LIN {X 0,Y 229.576,Z 730.403,A -85,B 0,C 180,E1 10386.317,E2 10386.317} C_VEL
LIN {X 0,Y 222.529,Z 739.722,A -85,B 0,C 180,E1 10381.712,E2 10381.712} C_VEL
LIN {X 0,Y 216.125,Z 748.376,A -85,B 0,C 180,E1 10376.069,E2 10376.069} C_VEL
LIN {X 0,Y 212.232,Z 754.139,A -85,B 0,C 180,E1 10371.117,E2 10371.117} C_VEL
LIN {X 0,Y 209.901,Z 758.178,A -85,B 0,C 180,E1 10366.605,E2 10366.605} C_VEL
LIN {X 0,Y 208.521,Z 761.292,A -85,B 0,C 180,E1 10361.898,E2 10361.898} C_VEL
LIN {X 0,Y 208.011,Z 763.279,A -85,B 0,C 180,E1 10357.456,E2 10357.456} C_VEL
LIN {X 0,Y 207.965,Z 764.362,A -85,B 0,C 180,E1 10353.031,E2 10353.031} C_VEL
LIN {X 0,Y 207.992,Z 764.571,A -85,B 0,C 180,E1 10348.898,E2 10348.898} C_VEL
LIN {X 0,Y 207.969,Z 763.727,A -85,B 0,C 180,E1 10343.929,E2 10343.929} C_VEL
LIN {X 0,Y 208.374,Z 761.739,A -85,B 0,C 180,E1 10338.935,E2 10338.935} C_VEL
LIN {X 0,Y 209.583,Z 758.806,A -85,B 0,C 180,E1 10334.223,E2 10334.223} C_VEL
LIN {X 0,Y 211.814,Z 754.811,A -85,B 0,C 180,E1 10329.557,E2 10329.557} C_VEL
LIN {X 0,Y 215.171,Z 749.706,A -85,B 0,C 180,E1 10324.98,E2 10324.98} C_VEL
LIN {X 0,Y 219.672,Z 743.459,A -85,B 0,C 180,E1 10320.559,E2 10320.559} C_VEL
LIN {X 0,Y 225.328,Z 735.97,A -85,B 0,C 180,E1 10316.316,E2 10316.316} C_VEL
LIN {X 0,Y 233.394,Z 725.524,A -85,B 0,C 180,E1 10311.603,E2 10311.603} C_VEL
LIN {X 0,Y 242.359,Z 713.434,A -85,B 0,C 180,E1 10307.428,E2 10307.428} C_VEL
LIN {X 0,Y 250.273,Z 702.419,A -85,B 0,C 180,E1 10304.353,E2 10304.353} C_VEL
LIN {X 0,Y 258.267,Z 690.731,A -85,B 0,C 180,E1 10301.66,E2 10301.66} C_VEL
LIN {X 0,Y 266.491,Z 677.953,A -85,B 0,C 180,E1 10299.223,E2 10299.223} C_VEL
LIN {X 0,Y 274.84,Z 663.987,A -85,B 0,C 180,E1 10297.018,E2 10297.018} C_VEL
LIN {X 0,Y 285.068,Z 645.138,A -85,B 0,C 180,E1 10294.627,E2 10294.627} C_VEL
LIN {X 0,Y 293.059,Z 628.408,A -85,B 0,C 180,E1 10292.943,E2 10292.943} C_VEL
LIN {X 0,Y 299.949,Z 612.279,A -85,B 0,C 180,E1 10291.614,E2 10291.614} C_VEL
LIN {X 0,Y 305.879,Z 596.561,A -85,B 0,C 180,E1 10290.544,E2 10290.544} C_VEL
LIN {X 0,Y 311.16,Z 580.497,A -85,B 0,C 180,E1 10289.644,E2 10289.644} C_VEL
LIN {X 0,Y 315.755,Z 564.123,A -85,B 0,C 180,E1 10288.9,E2 10288.9} C_VEL
LIN {X 0,Y 319.912,Z 546.219,A -85,B 0,C 180,E1 10288.263,E2 10288.263} C_VEL
LIN {X 0,Y 323.86,Z 523.655,A -85,B 0,C 180,E1 10287.653,E2 10287.653} C_VEL
LIN {X 0,Y 327.226,Z 489.016,A -85,B 0,C 180,E1 10286.991,E2 10286.991} C_VEL
LIN {X 0,Y 336.453,Z 381.786,A -85,B 0,C 180,E1 10285.079,E2 10285.079} C_VEL
LIN {X 0,Y 331.591,Z 370.301,A -85,B 0,C 180,E1 10282.611,E2 10282.611} C_VEL
LIN {X 0,Y 328.158,Z 363.719,A -85,B 0,C 180,E1 10280.745,E2 10280.745} C_VEL
LIN {X 0,Y 323.384,Z 355.371,A -85,B 0,C 180,E1 10277.825,E2 10277.825} C_VEL
LIN {X 0,Y 319.206,Z 348.74,A -85,B 0,C 180,E1 10274.791,E2 10274.791} C_VEL
LIN {X 0,Y 317.453,Z 345.951,A -85,B 0,C 180,E1 10273.293,E2 10273.293} C_VEL
LIN {X 0,Y 315.139,Z 342.181,A -85,B 0,C 180,E1 10270.975,E2 10270.975} C_VEL
LIN {X 0,Y 312.623,Z 337.855,A -85,B 0,C 180,E1 10267.628,E2 10267.628} C_VEL
LIN {X 0,Y 310.185,Z 334.373,A -85,B 0,C 180,E1 10260.369,E2 10260.369} C_VEL
LIN {X 0,Y 310.304,Z 334.935,A -85,B 0,C 180,E1 10257.784,E2 10257.784} C_VEL
LIN {X 0,Y 312.654,Z 337.983,A -85,B 0,C 180,E1 10252.003,E2 10252.003} C_VEL
LIN {X 0,Y 315.196,Z 342.253,A -85,B 0,C 180,E1 10248.657,E2 10248.657} C_VEL
LIN {X 0,Y 318.856,Z 348.121,A -85,B 0,C 180,E1 10245.192,E2 10245.192} C_VEL
LIN {X 0,Y 322.317,Z 353.748,A -85,B 0,C 180,E1 10242.581,E2 10242.581} C_VEL
LIN {X 0,Y 326.66,Z 361.098,A -85,B 0,C 180,E1 10239.811,E2 10239.811} C_VEL
LIN {X 0,Y 332.388,Z 371.39,A -85,B 0,C 180,E1 10236.698,E2 10236.698} C_VEL
LIN {X 0,Y 346.546,Z 396.133,A -85,B 0,C 180,E1 10230.674,E2 10230.674} C_VEL
LIN {X 0,Y 360.991,Z 413.89,A -85,B 0,C 180,E1 10226.169,E2 10226.169} C_VEL
LIN {X 0,Y 383.3,Z 434.199,A -85,B 0,C 180,E1 10220.855,E2 10220.855} C_VEL
LIN {X 0,Y 397.073,Z 444.864,A -85,B 0,C 180,E1 10218.092,E2 10218.092} C_VEL
LIN {X 0,Y 406.656,Z 452.456,A -85,B 0,C 180,E1 10216.052,E2 10216.052} C_VEL
LIN {X 0,Y 416.596,Z 460.43,A -85,B 0,C 180,E1 10213.743,E2 10213.743} C_VEL
LIN {X 0,Y 425.756,Z 468.037,A -85,B 0,C 180,E1 10211.379,E2 10211.379} C_VEL
LIN {X 0,Y 433.593,Z 474.542,A -85,B 0,C 180,E1 10209.181,E2 10209.181} C_VEL
LIN {X 0,Y 443.165,Z 482.341,A -85,B 0,C 180,E1 10206.343,E2 10206.343} C_VEL
LIN {X 0,Y 451.87,Z 489.268,A -85,B 0,C 180,E1 10203.637,E2 10203.637} C_VEL
LIN {X 0,Y 459.287,Z 495.387,A -85,B 0,C 180,E1 10201.176,E2 10201.176} C_VEL
LIN {X 0,Y 464.734,Z 499.578,A -85,B 0,C 180,E1 10199.269,E2 10199.269} C_VEL
LIN {X 0,Y 471.201,Z 504.679,A -85,B 0,C 180,E1 10196.867,E2 10196.867} C_VEL
LIN {X 0,Y 476.22,Z 508.342,A -85,B 0,C 180,E1 10194.9,E2 10194.9} C_VEL
LIN {X 0,Y 481.698,Z 512.833,A -85,B 0,C 180,E1 10192.524,E2 10192.524} C_VEL
LIN {X 0,Y 487.412,Z 516.593,A -85,B 0,C 180,E1 10189.844,E2 10189.844} C_VEL
LIN {X 0,Y 491.994,Z 520.595,A -85,B 0,C 180,E1 10187.38,E2 10187.38} C_VEL
LIN {X 0,Y 496.009,Z 523.409,A -85,B 0,C 180,E1 10184.951,E2 10184.951} C_VEL
LIN {X 0,Y 499.622,Z 525.352,A -85,B 0,C 180,E1 10182.41,E2 10182.41} C_VEL
LIN {X 0,Y 501.043,Z 526.363,A -85,B 0,C 180,E1 10181.276,E2 10181.276} C_VEL
LIN {X 0,Y 503.296,Z 528.639,A -85,B 0,C 180,E1 10179.029,E2 10179.029} C_VEL
LIN {X 0,Y 505.299,Z 530.408,A -85,B 0,C 180,E1 10176.59,E2 10176.59} C_VEL
LIN {X 0,Y 506.622,Z 531.453,A -85,B 0,C 180,E1 10174.074,E2 10174.074} C_VEL
LIN {X 0,Y 507.429,Z 531.971,A -85,B 0,C 180,E1 10171.468,E2 10171.468} C_VEL
LIN {X 0,Y 507.45,Z 531.985,A -85,B 0,C 180,E1 10169.097,E2 10169.097} C_VEL
LIN {X 0,Y 506.956,Z 531.659,A -85,B 0,C 180,E1 10166.608,E2 10166.608} C_VEL
LIN {X 0,Y 505.654,Z 530.72,A -85,B 0,C 180,E1 10164.068,E2 10164.068} C_VEL
LIN {X 0,Y 503.867,Z 529.16,A -85,B 0,C 180,E1 10161.557,E2 10161.557} C_VEL
LIN {X 0,Y 501.524,Z 526.933,A -85,B 0,C 180,E1 10159.2,E2 10159.2} C_VEL
LIN {X 0,Y 500.006,Z 525.51,A -85,B 0,C 180,E1 10157.881,E2 10157.881} C_VEL
LIN {X 0,Y 496.616,Z 523.748,A -85,B 0,C 180,E1 10155.425,E2 10155.425} C_VEL
LIN {X 0,Y 492.566,Z 521.055,A -85,B 0,C 180,E1 10152.963,E2 10152.963} C_VEL
LIN {X 0,Y 488.034,Z 517.174,A -85,B 0,C 180,E1 10150.469,E2 10150.469} C_VEL
LIN {X 0,Y 484.075,Z 514.456,A -85,B 0,C 180,E1 10148.558,E2 10148.558} C_VEL
LIN {X 0,Y 478.527,Z 510.37,A -85,B 0,C 180,E1 10146.089,E2 10146.089} C_VEL
LIN {X 0,Y 473.228,Z 506.031,A -85,B 0,C 180,E1 10143.895,E2 10143.895} C_VEL
LIN {X 0,Y 466.718,Z 501.246,A -85,B 0,C 180,E1 10141.448,E2 10141.448} C_VEL
LIN {X 0,Y 461.036,Z 496.657,A -85,B 0,C 180,E1 10139.431,E2 10139.431} C_VEL
LIN {X 0,Y 453.633,Z 490.858,A -85,B 0,C 180,E1 10136.95,E2 10136.95} C_VEL
LIN {X 0,Y 446.485,Z 485.103,A -85,B 0,C 180,E1 10134.678,E2 10134.678} C_VEL
LIN {X 0,Y 437.683,Z 477.869,A -85,B 0,C 180,E1 10132.014,E2 10132.014} C_VEL
LIN {X 0,Y 428.629,Z 470.268,A -85,B 0,C 180,E1 10129.402,E2 10129.402} C_VEL
LIN {X 0,Y 420.998,Z 464.055,A -85,B 0,C 180,E1 10127.364,E2 10127.364} C_VEL
LIN {X 0,Y 411.623,Z 456.502,A -85,B 0,C 180,E1 10125.08,E2 10125.08} C_VEL
LIN {X 0,Y 401.509,Z 448.491,A -85,B 0,C 180,E1 10122.833,E2 10122.833} C_VEL
LIN {X 0,Y 390.28,Z 439.766,A -85,B 0,C 180,E1 10120.55,E2 10120.55} C_VEL
LIN {X 0,Y 363.524,Z 416.49,A -85,B 0,C 180,E1 10114.514,E2 10114.514} C_VEL
LIN {X 0,Y 349.69,Z 400.357,A -85,B 0,C 180,E1 10110.405,E2 10110.405} C_VEL
LIN {X 0,Y 339.201,Z 384.437,A -85,B 0,C 180,E1 10106.478,E2 10106.478} C_VEL
LIN {X 0,Y 331.747,Z 370.145,A -85,B 0,C 180,E1 10102.974,E2 10102.974} C_VEL
LIN {X 0,Y 325.408,Z 358.84,A -85,B 0,C 180,E1 10099.428,E2 10099.428} C_VEL
LIN {X 0,Y 320.76,Z 351.104,A -85,B 0,C 180,E1 10096.293,E2 10096.293} C_VEL
LIN {X 0,Y 317.522,Z 346.047,A -85,B 0,C 180,E1 10093.661,E2 10093.661} C_VEL
LIN {X 0,Y 315.196,Z 342.25,A -85,B 0,C 180,E1 10091.343,E2 10091.343} C_VEL
LIN {X 0,Y 312.654,Z 337.981,A -85,B 0,C 180,E1 10087.997,E2 10087.997} C_VEL
LIN {X 0,Y 310.184,Z 334.34,A -85,B 0,C 180,E1 10080.554,E2 10080.554} C_VEL
LIN {X 0,Y 310.42,Z 335.246,A -85,B 0,C 180,E1 10077.415,E2 10077.415} C_VEL
LIN {X 0,Y 312.674,Z 338,A -85,B 0,C 180,E1 10072.281,E2 10072.281} C_VEL
LIN {X 0,Y 315.139,Z 342.183,A -85,B 0,C 180,E1 10069.025,E2 10069.025} C_VEL
LIN {X 0,Y 318.785,Z 347.988,A -85,B 0,C 180,E1 10065.56,E2 10065.56} C_VEL
LIN {X 0,Y 322.733,Z 354.42,A -85,B 0,C 180,E1 10062.604,E2 10062.604} C_VEL
LIN {X 0,Y 327.577,Z 362.616,A -85,B 0,C 180,E1 10059.59,E2 10059.59} C_VEL
LIN {X 0,Y 331.359,Z 369.794,A -85,B 0,C 180,E1 10057.513,E2 10057.513} C_VEL
LIN {X 0,Y 335.907,Z 380.499,A -85,B 0,C 180,E1 10055.183,E2 10055.183} C_VEL
LIN {X 0,Y 336.48,Z 382.275,A -85,B 0,C 180,E1 10054.888,E2 10054.888} C_VEL
LIN {X 0,Y 324.566,Z 517.418,A -85,B 0,C 180,E1 10052.477,E2 10052.477} C_VEL
LIN {X 0,Y 321.459,Z 538.537,A -85,B 0,C 180,E1 10051.966,E2 10051.966} C_VEL
LIN {X 0,Y 316.405,Z 561.647,A -85,B 0,C 180,E1 10051.199,E2 10051.199} C_VEL
LIN {X 0,Y 311.542,Z 579.253,A -85,B 0,C 180,E1 10050.418,E2 10050.418} C_VEL
LIN {X 0,Y 306.252,Z 595.5,A -85,B 0,C 180,E1 10049.522,E2 10049.522} C_VEL
LIN {X 0,Y 300.315,Z 611.359,A -85,B 0,C 180,E1 10048.455,E2 10048.455} C_VEL
LIN {X 0,Y 300.203,Z 611.641,A -85,B 0,C 180,E1 10048.434,E2 10048.434} C_VEL
LIN {X 0,Y 296.909,Z 618.594,A -85,B 0,C 180,E1 10048.072,E2 10048.072} C_VEL
LIN {X 0,Y 285.993,Z 635.3,A -85,B 0,C 180,E1 10047.577,E2 10047.577} C_VEL
LIN {X 0,Y 282.279,Z 641.505,A -85,B 0,C 180,E1 10047.099,E2 10047.099} C_VEL
LIN {X 0,Y 273.798,Z 657.322,A -85,B 0,C 180,E1 10045.242,E2 10045.242} C_VEL
LIN {X 0,Y 263.053,Z 675.28,A -85,B 0,C 180,E1 10042.591,E2 10042.591} C_VEL
LIN {X 0,Y 254.155,Z 688.774,A -85,B 0,C 180,E1 10040.09,E2 10040.09} C_VEL
LIN {X 0,Y 245.788,Z 700.659,A -85,B 0,C 180,E1 10037.411,E2 10037.411} C_VEL
LIN {X 0,Y 237.997,Z 711.151,A -85,B 0,C 180,E1 10034.549,E2 10034.549} C_VEL
LIN {X 0,Y 230.344,Z 721.041,A -85,B 0,C 180,E1 10031.278,E2 10031.278} C_VEL
LIN {X 0,Y 223.04,Z 730.224,A -85,B 0,C 180,E1 10027.561,E2 10027.561} C_VEL
LIN {X 0,Y 215.613,Z 739.544,A -85,B 0,C 180,E1 10022.854,E2 10022.854} C_VEL
LIN {X 0,Y 208.793,Z 748.224,A -85,B 0,C 180,E1 10017.033,E2 10017.033} C_VEL
LIN {X 0,Y 204.742,Z 753.82,A -85,B 0,C 180,E1 10012.085,E2 10012.085} C_VEL
LIN {X 0,Y 202.12,Z 758,A -85,B 0,C 180,E1 10007.264,E2 10007.264} C_VEL
LIN {X 0,Y 200.59,Z 761.149,A -85,B 0,C 180,E1 10002.308,E2 10002.308} C_VEL
LIN {X 0,Y 200.012,Z 763.193,A -85,B 0,C 180,E1 9997.467,E2 9997.467} C_VEL
LIN {X 0,Y 199.965,Z 764.187,A -85,B 0,C 180,E1 9993.153,E2 9993.153} C_VEL
LIN {X 0,Y 199.993,Z 764.396,A -85,B 0,C 180,E1 9988.854,E2 9988.854} C_VEL
LIN {X 0,Y 199.969,Z 763.641,A -85,B 0,C 180,E1 9983.973,E2 9983.973} C_VEL
LIN {X 0,Y 200.391,Z 761.712,A -85,B 0,C 180,E1 9978.78,E2 9978.78} C_VEL
LIN {X 0,Y 201.775,Z 758.628,A -85,B 0,C 180,E1 9973.595,E2 9973.595} C_VEL
LIN {X 0,Y 204.194,Z 754.633,A -85,B 0,C 180,E1 9968.758,E2 9968.758} C_VEL
LIN {X 0,Y 207.791,Z 749.536,A -85,B 0,C 180,E1 9964.034,E2 9964.034} C_VEL
LIN {X 0,Y 212.273,Z 743.68,A -85,B 0,C 180,E1 9959.739,E2 9959.739} C_VEL
LIN {X 0,Y 217.804,Z 736.729,A -85,B 0,C 180,E1 9955.626,E2 9955.626} C_VEL
LIN {X 0,Y 224.59,Z 728.288,A -85,B 0,C 180,E1 9951.589,E2 9951.589} C_VEL
LIN {X 0,Y 233.32,Z 717.328,A -85,B 0,C 180,E1 9947.389,E2 9947.389} C_VEL
LIN {X 0,Y 243.507,Z 703.824,A -85,B 0,C 180,E1 9943.39,E2 9943.39} C_VEL
LIN {X 0,Y 252.319,Z 691.443,A -85,B 0,C 180,E1 9940.469,E2 9940.469} C_VEL
LIN {X 0,Y 260.46,Z 679.274,A -85,B 0,C 180,E1 9938.106,E2 9938.106} C_VEL
LIN {X 0,Y 268.349,Z 666.612,A -85,B 0,C 180,E1 9936.055,E2 9936.055} C_VEL
LIN {X 0,Y 276.069,Z 653.203,A -85,B 0,C 180,E1 9934.244,E2 9934.244} C_VEL
LIN {X 0,Y 283.669,Z 638.754,A -85,B 0,C 180,E1 9932.614,E2 9932.614} C_VEL
LIN {X 0,Y 291.329,Z 622.592,A -85,B 0,C 180,E1 9931.106,E2 9931.106} C_VEL
LIN {X 0,Y 299.967,Z 601.695,A -85,B 0,C 180,E1 9929.555,E2 9929.555} C_VEL
LIN {X 0,Y 306.486,Z 582.805,A -85,B 0,C 180,E1 9928.465,E2 9928.465} C_VEL
LIN {X 0,Y 311.362,Z 566.176,A -85,B 0,C 180,E1 9927.699,E2 9927.699} C_VEL
LIN {X 0,Y 315.623,Z 548.674,A -85,B 0,C 180,E1 9927.066,E2 9927.066} C_VEL
LIN {X 0,Y 318.97,Z 531.138,A -85,B 0,C 180,E1 9926.574,E2 9926.574} C_VEL
LIN {X 0,Y 321.456,Z 512.557,A -85,B 0,C 180,E1 9926.159,E2 9926.159} C_VEL
LIN {X 0,Y 332.773,Z 385.796,A -85,B 0,C 180,E1 9923.908,E2 9923.908} C_VEL
LIN {X 0,Y 328.392,Z 375.154,A -85,B 0,C 180,E1 9921.525,E2 9921.525} C_VEL
LIN {X 0,Y 323.343,Z 365.828,A -85,B 0,C 180,E1 9918.526,E2 9918.526} C_VEL
LIN {X 0,Y 318.985,Z 358.378,A -85,B 0,C 180,E1 9915.453,E2 9915.453} C_VEL
LIN {X 0,Y 316.074,Z 353.64,A -85,B 0,C 180,E1 9912.98,E2 9912.98} C_VEL
LIN {X 0,Y 313.829,Z 349.888,A -85,B 0,C 180,E1 9910.649,E2 9910.649} C_VEL
LIN {X 0,Y 311.244,Z 345.447,A -85,B 0,C 180,E1 9907.012,E2 9907.012} C_VEL
LIN {X 0,Y 309.204,Z 342.3,A -85,B 0,C 180,E1 9900.185,E2 9900.185} C_VEL
LIN {X 0,Y 309.417,Z 343.167,A -85,B 0,C 180,E1 9897.222,E2 9897.222} C_VEL
LIN {X 0,Y 311.549,Z 345.958,A -85,B 0,C 180,E1 9892.16,E2 9892.16} C_VEL
LIN {X 0,Y 314.625,Z 351.207,A -85,B 0,C 180,E1 9888.162,E2 9888.162} C_VEL
LIN {X 0,Y 317.538,Z 356.047,A -85,B 0,C 180,E1 9885.409,E2 9885.409} C_VEL
LIN {X 0,Y 320.818,Z 361.511,A -85,B 0,C 180,E1 9882.871,E2 9882.871} C_VEL
LIN {X 0,Y 325.497,Z 369.707,A -85,B 0,C 180,E1 9879.829,E2 9879.829} C_VEL
LIN {X 0,Y 331.416,Z 380.885,A -85,B 0,C 180,E1 9876.578,E2 9876.578} C_VEL
LIN {X 0,Y 342.541,Z 401.036,A -85,B 0,C 180,E1 9871.683,E2 9871.683} C_VEL
LIN {X 0,Y 356.013,Z 418.443,A -85,B 0,C 180,E1 9867.224,E2 9867.224} C_VEL
LIN {X 0,Y 373.061,Z 435.003,A -85,B 0,C 180,E1 9862.815,E2 9862.815} C_VEL
LIN {X 0,Y 393.784,Z 451.72,A -85,B 0,C 180,E1 9858.492,E2 9858.492} C_VEL
LIN {X 0,Y 404.068,Z 459.754,A -85,B 0,C 180,E1 9856.338,E2 9856.338} C_VEL
LIN {X 0,Y 413.478,Z 467.249,A -85,B 0,C 180,E1 9854.192,E2 9854.192} C_VEL
LIN {X 0,Y 422.851,Z 474.87,A -85,B 0,C 180,E1 9851.853,E2 9851.853} C_VEL
LIN {X 0,Y 431.409,Z 481.9,A -85,B 0,C 180,E1 9849.484,E2 9849.484} C_VEL
LIN {X 0,Y 441.106,Z 489.743,A -85,B 0,C 180,E1 9846.636,E2 9846.636} C_VEL
LIN {X 0,Y 449.6,Z 496.451,A -85,B 0,C 180,E1 9844.006,E2 9844.006} C_VEL
LIN {X 0,Y 457.074,Z 502.656,A -85,B 0,C 180,E1 9841.551,E2 9841.551} C_VEL
LIN {X 0,Y 463.048,Z 507.191,A -85,B 0,C 180,E1 9839.49,E2 9839.49} C_VEL
LIN {X 0,Y 469.743,Z 512.437,A -85,B 0,C 180,E1 9837.026,E2 9837.026} C_VEL
LIN {X 0,Y 474.826,Z 516.148,A -85,B 0,C 180,E1 9835.037,E2 9835.037} C_VEL
LIN {X 0,Y 480.395,Z 520.663,A -85,B 0,C 180,E1 9832.644,E2 9832.644} C_VEL
LIN {X 0,Y 486.164,Z 524.446,A -85,B 0,C 180,E1 9829.96,E2 9829.96} C_VEL
LIN {X 0,Y 490.743,Z 528.395,A -85,B 0,C 180,E1 9827.531,E2 9827.531} C_VEL
LIN {X 0,Y 494.745,Z 531.223,A -85,B 0,C 180,E1 9825.11,E2 9825.11} C_VEL
LIN {X 0,Y 498.505,Z 533.242,A -85,B 0,C 180,E1 9822.509,E2 9822.509} C_VEL
LIN {X 0,Y 500.029,Z 534.336,A -85,B 0,C 180,E1 9821.3,E2 9821.3} C_VEL
LIN {X 0,Y 502.292,Z 536.591,A -85,B 0,C 180,E1 9819.047,E2 9819.047} C_VEL
LIN {X 0,Y 504.312,Z 538.351,A -85,B 0,C 180,E1 9816.602,E2 9816.602} C_VEL
LIN {X 0,Y 505.641,Z 539.394,A -85,B 0,C 180,E1 9814.082,E2 9814.082} C_VEL
LIN {X 0,Y 506.453,Z 539.911,A -85,B 0,C 180,E1 9811.471,E2 9811.471} C_VEL
LIN {X 0,Y 506.474,Z 539.925,A -85,B 0,C 180,E1 9809.095,E2 9809.095} C_VEL
LIN {X 0,Y 505.979,Z 539.6,A -85,B 0,C 180,E1 9806.602,E2 9806.602} C_VEL
LIN {X 0,Y 504.686,Z 538.676,A -85,B 0,C 180,E1 9804.088,E2 9804.088} C_VEL
LIN {X 0,Y 502.973,Z 537.211,A -85,B 0,C 180,E1 9801.657,E2 9801.657} C_VEL
LIN {X 0,Y 500.51,Z 534.898,A -85,B 0,C 180,E1 9799.178,E2 9799.178} C_VEL
LIN {X 0,Y 498.821,Z 533.377,A -85,B 0,C 180,E1 9797.734,E2 9797.734} C_VEL
LIN {X 0,Y 495.316,Z 531.539,A -85,B 0,C 180,E1 9795.23,E2 9795.23} C_VEL
LIN {X 0,Y 491.354,Z 528.893,A -85,B 0,C 180,E1 9792.841,E2 9792.841} C_VEL
LIN {X 0,Y 486.699,Z 524.95,A -85,B 0,C 180,E1 9790.313,E2 9790.313} C_VEL
LIN {X 0,Y 481.953,Z 521.71,A -85,B 0,C 180,E1 9788.03,E2 9788.03} C_VEL
LIN {X 0,Y 476.405,Z 517.535,A -85,B 0,C 180,E1 9785.629,E2 9785.629} C_VEL
LIN {X 0,Y 471.685,Z 513.736,A -85,B 0,C 180,E1 9783.706,E2 9783.706} C_VEL
LIN {X 0,Y 465.205,Z 508.978,A -85,B 0,C 180,E1 9781.275,E2 9781.275} C_VEL
LIN {X 0,Y 459.27,Z 504.242,A -85,B 0,C 180,E1 9779.191,E2 9779.191} C_VEL
LIN {X 0,Y 451.846,Z 498.442,A -85,B 0,C 180,E1 9776.721,E2 9776.721} C_VEL
LIN {X 0,Y 443.612,Z 491.846,A -85,B 0,C 180,E1 9774.13,E2 9774.13} C_VEL
LIN {X 0,Y 435.125,Z 484.929,A -85,B 0,C 180,E1 9771.591,E2 9771.591} C_VEL
LIN {X 0,Y 426.196,Z 477.515,A -85,B 0,C 180,E1 9769.064,E2 9769.064} C_VEL
LIN {X 0,Y 418.744,Z 471.473,A -85,B 0,C 180,E1 9767.094,E2 9767.094} C_VEL
LIN {X 0,Y 408.582,Z 463.367,A -85,B 0,C 180,E1 9764.666,E2 9764.666} C_VEL
LIN {X 0,Y 398.159,Z 455.228,A -85,B 0,C 180,E1 9762.408,E2 9762.408} C_VEL
LIN {X 0,Y 385.414,Z 445.344,A -85,B 0,C 180,E1 9759.852,E2 9759.852} C_VEL
LIN {X 0,Y 360.455,Z 423.252,A -85,B 0,C 180,E1 9754.032,E2 9754.032} C_VEL
LIN {X 0,Y 346.851,Z 407.086,A -85,B 0,C 180,E1 9749.868,E2 9749.868} C_VEL
LIN {X 0,Y 336.504,Z 391.004,A -85,B 0,C 180,E1 9745.852,E2 9745.852} C_VEL
LIN {X 0,Y 329.357,Z 376.881,A -85,B 0,C 180,E1 9742.349,E2 9742.349} C_VEL
LIN {X 0,Y 323.439,Z 365.989,A -85,B 0,C 180,E1 9738.895,E2 9738.895} C_VEL
LIN {X 0,Y 319.067,Z 358.487,A -85,B 0,C 180,E1 9735.821,E2 9735.821} C_VEL
LIN {X 0,Y 315.948,Z 353.458,A -85,B 0,C 180,E1 9733.171,E2 9733.171} C_VEL
LIN {X 0,Y 313.885,Z 349.959,A -85,B 0,C 180,E1 9731.019,E2 9731.019} C_VEL
LIN {X 0,Y 311.282,Z 345.481,A -85,B 0,C 180,E1 9727.382,E2 9727.382} C_VEL
LIN {X 0,Y 309.204,Z 342.276,A -85,B 0,C 180,E1 9720.37,E2 9720.37} C_VEL
LIN {X 0,Y 309.521,Z 343.402,A -85,B 0,C 180,E1 9717.037,E2 9717.037} C_VEL
LIN {X 0,Y 311.518,Z 345.832,A -85,B 0,C 180,E1 9712.531,E2 9712.531} C_VEL
LIN {X 0,Y 313.996,Z 350.073,A -85,B 0,C 180,E1 9709.171,E2 9709.171} C_VEL
LIN {X 0,Y 317.365,Z 355.729,A -85,B 0,C 180,E1 9705.867,E2 9705.867} C_VEL
LIN {X 0,Y 321.608,Z 362.734,A -85,B 0,C 180,E1 9702.634,E2 9702.634} C_VEL
LIN {X 0,Y 326.414,Z 371.468,A -85,B 0,C 180,E1 9699.591,E2 9699.591} C_VEL
LIN {X 0,Y 329.354,Z 377.369,A -85,B 0,C 180,E1 9697.933,E2 9697.933} C_VEL
LIN {X 0,Y 332.795,Z 386.105,A -85,B 0,C 180,E1 9696.068,E2 9696.068} C_VEL
LIN {X 0,Y 320.935,Z 517.284,A -85,B 0,C 180,E1 9693.746,E2 9693.746} C_VEL
LIN {X 0,Y 317.72,Z 538.657,A -85,B 0,C 180,E1 9693.235,E2 9693.235} C_VEL
LIN {X 0,Y 312.796,Z 560.808,A -85,B 0,C 180,E1 9692.513,E2 9692.513} C_VEL
LIN {X 0,Y 307.654,Z 579.077,A -85,B 0,C 180,E1 9691.72,E2 9691.72} C_VEL
LIN {X 0,Y 302.248,Z 595.324,A -85,B 0,C 180,E1 9690.837,E2 9690.837} C_VEL
LIN {X 0,Y 296.176,Z 611.183,A -85,B 0,C 180,E1 9689.784,E2 9689.784} C_VEL
LIN {X 0,Y 289.48,Z 626.62,A -85,B 0,C 180,E1 9688.544,E2 9688.544} C_VEL
LIN {X 0,Y 282.279,Z 641.505,A -85,B 0,C 180,E1 9687.099,E2 9687.099} C_VEL
LIN {X 0,Y 278.481,Z 647.851,A -85,B 0,C 180,E1 9686.583,E2 9686.583} C_VEL
LIN {X 0,Y 266.227,Z 663.246,A -85,B 0,C 180,E1 9685.662,E2 9685.662} C_VEL
LIN {X 0,Y 262.112,Z 668.947,A -85,B 0,C 180,E1 9684.998,E2 9684.998} C_VEL
LIN {X 0,Y 250.948,Z 685.928,A -85,B 0,C 180,E1 9682.075,E2 9682.075} C_VEL
LIN {X 0,Y 240.863,Z 699.801,A -85,B 0,C 180,E1 9679.012,E2 9679.012} C_VEL
LIN {X 0,Y 232.81,Z 710.272,A -85,B 0,C 180,E1 9676.173,E2 9676.173} C_VEL
LIN {X 0,Y 224.775,Z 720.244,A -85,B 0,C 180,E1 9672.884,E2 9672.884} C_VEL
LIN {X 0,Y 217.519,Z 728.962,A -85,B 0,C 180,E1 9669.366,E2 9669.366} C_VEL
LIN {X 0,Y 210.707,Z 737.02,A -85,B 0,C 180,E1 9665.37,E2 9665.37} C_VEL
LIN {X 0,Y 204.595,Z 744.302,A -85,B 0,C 180,E1 9660.869,E2 9660.869} C_VEL
LIN {X 0,Y 198.742,Z 751.699,A -85,B 0,C 180,E1 9654.996,E2 9654.996} C_VEL
LIN {X 0,Y 194.638,Z 757.403,A -85,B 0,C 180,E1 9648.57,E2 9648.57} C_VEL
LIN {X 0,Y 192.77,Z 760.789,A -85,B 0,C 180,E1 9643.191,E2 9643.191} C_VEL
LIN {X 0,Y 192.048,Z 762.927,A -85,B 0,C 180,E1 9638.08,E2 9638.08} C_VEL
LIN {X 0,Y 191.965,Z 764.012,A -85,B 0,C 180,E1 9633.284,E2 9633.284} C_VEL
LIN {X 0,Y 191.994,Z 764.221,A -85,B 0,C 180,E1 9628.806,E2 9628.806} C_VEL
LIN {X 0,Y 191.975,Z 763.465,A -85,B 0,C 180,E1 9623.721,E2 9623.721} C_VEL
LIN {X 0,Y 192.46,Z 761.535,A -85,B 0,C 180,E1 9618.312,E2 9618.312} C_VEL
LIN {X 0,Y 193.991,Z 758.451,A -85,B 0,C 180,E1 9612.917,E2 9612.917} C_VEL
LIN {X 0,Y 196.615,Z 754.455,A -85,B 0,C 180,E1 9607.897,E2 9607.897} C_VEL
LIN {X 0,Y 200.477,Z 749.357,A -85,B 0,C 180,E1 9603.012,E2 9603.012} C_VEL
LIN {X 0,Y 205.587,Z 743.101,A -85,B 0,C 180,E1 9598.319,E2 9598.319} C_VEL
LIN {X 0,Y 211.908,Z 735.613,A -85,B 0,C 180,E1 9593.862,E2 9593.862} C_VEL
LIN {X 0,Y 220.815,Z 725.167,A -85,B 0,C 180,E1 9588.967,E2 9588.967} C_VEL
LIN {X 0,Y 230.596,Z 713.077,A -85,B 0,C 180,E1 9584.682,E2 9584.682} C_VEL
LIN {X 0,Y 239.154,Z 702.063,A -85,B 0,C 180,E1 9581.558,E2 9581.558} C_VEL
LIN {X 0,Y 247.742,Z 690.376,A -85,B 0,C 180,E1 9578.845,E2 9578.845} C_VEL
LIN {X 0,Y 256.188,Z 678.097,A -85,B 0,C 180,E1 9576.496,E2 9576.496} C_VEL
LIN {X 0,Y 264.691,Z 664.753,A -85,B 0,C 180,E1 9574.382,E2 9574.382} C_VEL
LIN {X 0,Y 274.284,Z 648.326,A -85,B 0,C 180,E1 9572.26,E2 9572.26} C_VEL
LIN {X 0,Y 284.083,Z 629.165,A -85,B 0,C 180,E1 9570.31,E2 9570.31} C_VEL
LIN {X 0,Y 291.437,Z 612.846,A -85,B 0,C 180,E1 9568.984,E2 9568.984} C_VEL
LIN {X 0,Y 297.877,Z 596.594,A -85,B 0,C 180,E1 9567.9,E2 9567.9} C_VEL
LIN {X 0,Y 303.532,Z 580.144,A -85,B 0,C 180,E1 9567.006,E2 9567.006} C_VEL
LIN {X 0,Y 308.317,Z 563.772,A -85,B 0,C 180,E1 9566.288,E2 9566.288} C_VEL
LIN {X 0,Y 312.637,Z 545.869,A -85,B 0,C 180,E1 9565.673,E2 9565.673} C_VEL
LIN {X 0,Y 316.735,Z 523.304,A -85,B 0,C 180,E1 9565.082,E2 9565.082} C_VEL
LIN {X 0,Y 320.266,Z 488.665,A -85,B 0,C 180,E1 9564.433,E2 9564.433} C_VEL
LIN {X 0,Y 329.201,Z 389.682,A -85,B 0,C 180,E1 9562.69,E2 9562.69} C_VEL
LIN {X 0,Y 325.426,Z 380.55,A -85,B 0,C 180,E1 9560.504,E2 9560.504} C_VEL
LIN {X 0,Y 320.388,Z 371.156,A -85,B 0,C 180,E1 9557.289,E2 9557.289} C_VEL
LIN {X 0,Y 316.774,Z 364.905,A -85,B 0,C 180,E1 9554.533,E2 9554.533} C_VEL
LIN {X 0,Y 314.518,Z 361.051,A -85,B 0,C 180,E1 9552.485,E2 9552.485} C_VEL
LIN {X 0,Y 312.53,Z 357.593,A -85,B 0,C 180,E1 9550.321,E2 9550.321} C_VEL
LIN {X 0,Y 310.159,Z 353.333,A -85,B 0,C 180,E1 9546.851,E2 9546.851} C_VEL
LIN {X 0,Y 308.229,Z 350.242,A -85,B 0,C 180,E1 9540.186,E2 9540.186} C_VEL
LIN {X 0,Y 308.439,Z 351.139,A -85,B 0,C 180,E1 9537.213,E2 9537.213} C_VEL
LIN {X 0,Y 310.399,Z 353.786,A -85,B 0,C 180,E1 9532.411,E2 9532.411} C_VEL
LIN {X 0,Y 313.291,Z 358.897,A -85,B 0,C 180,E1 9528.494,E2 9528.494} C_VEL
LIN {X 0,Y 316.025,Z 363.597,A -85,B 0,C 180,E1 9525.806,E2 9525.806} C_VEL
LIN {X 0,Y 319.817,Z 370.047,A -85,B 0,C 180,E1 9522.816,E2 9522.816} C_VEL
LIN {X 0,Y 324.45,Z 378.795,A -85,B 0,C 180,E1 9519.761,E2 9519.761} C_VEL
LIN {X 0,Y 329.39,Z 388.426,A -85,B 0,C 180,E1 9516.994,E2 9516.994} C_VEL
LIN {X 0,Y 339.726,Z 407.61,A -85,B 0,C 180,E1 9512.288,E2 9512.288} C_VEL
LIN {X 0,Y 352.804,Z 424.901,A -85,B 0,C 180,E1 9507.804,E2 9507.804} C_VEL
LIN {X 0,Y 369.71,Z 441.689,A -85,B 0,C 180,E1 9503.295,E2 9503.295} C_VEL
LIN {X 0,Y 391.486,Z 459.303,A -85,B 0,C 180,E1 9498.682,E2 9498.682} C_VEL
LIN {X 0,Y 401.904,Z 467.355,A -85,B 0,C 180,E1 9496.536,E2 9496.536} C_VEL
LIN {X 0,Y 411.921,Z 475.253,A -85,B 0,C 180,E1 9494.268,E2 9494.268} C_VEL
LIN {X 0,Y 421.104,Z 482.678,A -85,B 0,C 180,E1 9491.995,E2 9491.995} C_VEL
LIN {X 0,Y 430.213,Z 490.096,A -85,B 0,C 180,E1 9489.5,E2 9489.5} C_VEL
LIN {X 0,Y 439.479,Z 497.538,A -85,B 0,C 180,E1 9486.787,E2 9486.787} C_VEL
LIN {X 0,Y 447.767,Z 504.021,A -85,B 0,C 180,E1 9484.239,E2 9484.239} C_VEL
LIN {X 0,Y 455.265,Z 510.219,A -85,B 0,C 180,E1 9481.792,E2 9481.792} C_VEL
LIN {X 0,Y 461.595,Z 515.003,A -85,B 0,C 180,E1 9479.63,E2 9479.63} C_VEL
LIN {X 0,Y 468.288,Z 520.194,A -85,B 0,C 180,E1 9477.185,E2 9477.185} C_VEL
LIN {X 0,Y 473.405,Z 523.934,A -85,B 0,C 180,E1 9475.185,E2 9475.185} C_VEL
LIN {X 0,Y 479.17,Z 528.547,A -85,B 0,C 180,E1 9472.731,E2 9472.731} C_VEL
LIN {X 0,Y 484.917,Z 532.299,A -85,B 0,C 180,E1 9470.076,E2 9470.076} C_VEL
LIN {X 0,Y 489.404,Z 536.137,A -85,B 0,C 180,E1 9467.721,E2 9467.721} C_VEL
LIN {X 0,Y 493.485,Z 539.036,A -85,B 0,C 180,E1 9465.27,E2 9465.27} C_VEL
LIN {X 0,Y 497.33,Z 541.103,A -85,B 0,C 180,E1 9462.657,E2 9462.657} C_VEL
LIN {X 0,Y 499.016,Z 542.307,A -85,B 0,C 180,E1 9461.323,E2 9461.323} C_VEL
LIN {X 0,Y 501.398,Z 544.648,A -85,B 0,C 180,E1 9458.947,E2 9458.947} C_VEL
LIN {X 0,Y 503.387,Z 546.35,A -85,B 0,C 180,E1 9456.5,E2 9456.5} C_VEL
LIN {X 0,Y 504.659,Z 547.335,A -85,B 0,C 180,E1 9454.09,E2 9454.09} C_VEL
LIN {X 0,Y 505.478,Z 547.844,A -85,B 0,C 180,E1 9451.587,E2 9451.587} C_VEL
LIN {X 0,Y 505.497,Z 547.865,A -85,B 0,C 180,E1 9449.093,E2 9449.093} C_VEL
LIN {X 0,Y 505,Z 547.54,A -85,B 0,C 180,E1 9446.595,E2 9446.595} C_VEL
LIN {X 0,Y 503.7,Z 546.618,A -85,B 0,C 180,E1 9444.076,E2 9444.076} C_VEL
LIN {X 0,Y 501.857,Z 545.063,A -85,B 0,C 180,E1 9441.523,E2 9441.523} C_VEL
LIN {X 0,Y 499.496,Z 542.861,A -85,B 0,C 180,E1 9439.156,E2 9439.156} C_VEL
LIN {X 0,Y 497.616,Z 541.232,A -85,B 0,C 180,E1 9437.568,E2 9437.568} C_VEL
LIN {X 0,Y 493.864,Z 539.254,A -85,B 0,C 180,E1 9434.961,E2 9434.961} C_VEL
LIN {X 0,Y 489.856,Z 536.497,A -85,B 0,C 180,E1 9432.542,E2 9432.542} C_VEL
LIN {X 0,Y 485.314,Z 532.676,A -85,B 0,C 180,E1 9430.129,E2 9430.129} C_VEL
LIN {X 0,Y 480.246,Z 529.276,A -85,B 0,C 180,E1 9427.736,E2 9427.736} C_VEL
LIN {X 0,Y 474.652,Z 524.989,A -85,B 0,C 180,E1 9425.315,E2 9425.315} C_VEL
LIN {X 0,Y 469.995,Z 521.356,A -85,B 0,C 180,E1 9423.468,E2 9423.468} C_VEL
LIN {X 0,Y 463.441,Z 516.539,A -85,B 0,C 180,E1 9421.031,E2 9421.031} C_VEL
LIN {X 0,Y 457.074,Z 511.512,A -85,B 0,C 180,E1 9418.799,E2 9418.799} C_VEL
LIN {X 0,Y 449.615,Z 505.647,A -85,B 0,C 180,E1 9416.349,E2 9416.349} C_VEL
LIN {X 0,Y 440.169,Z 498.116,A -85,B 0,C 180,E1 9413.419,E2 9413.419} C_VEL
LIN {X 0,Y 431.861,Z 491.441,A -85,B 0,C 180,E1 9410.974,E2 9410.974} C_VEL
LIN {X 0,Y 422.333,Z 483.62,A -85,B 0,C 180,E1 9408.318,E2 9408.318} C_VEL
LIN {X 0,Y 413.491,Z 476.411,A -85,B 0,C 180,E1 9406.105,E2 9406.105} C_VEL
LIN {X 0,Y 404.534,Z 469.435,A -85,B 0,C 180,E1 9404.041,E2 9404.041} C_VEL
LIN {X 0,Y 393.56,Z 460.97,A -85,B 0,C 180,E1 9401.732,E2 9401.732} C_VEL
LIN {X 0,Y 371.502,Z 443.253,A -85,B 0,C 180,E1 9397.126,E2 9397.126} C_VEL
LIN {X 0,Y 353.634,Z 425.879,A -85,B 0,C 180,E1 9392.447,E2 9392.447} C_VEL
LIN {X 0,Y 340.122,Z 408.228,A -85,B 0,C 180,E1 9387.868,E2 9387.868} C_VEL
LIN {X 0,Y 330.1,Z 389.934,A -85,B 0,C 180,E1 9383.379,E2 9383.379} C_VEL
LIN {X 0,Y 325.165,Z 380.117,A -85,B 0,C 180,E1 9380.662,E2 9380.662} C_VEL
LIN {X 0,Y 320.297,Z 370.994,A -85,B 0,C 180,E1 9377.533,E2 9377.533} C_VEL
LIN {X 0,Y 316.744,Z 364.85,A -85,B 0,C 180,E1 9374.815,E2 9374.815} C_VEL
LIN {X 0,Y 314.399,Z 360.867,A -85,B 0,C 180,E1 9372.676,E2 9372.676} C_VEL
LIN {X 0,Y 312.585,Z 357.666,A -85,B 0,C 180,E1 9370.692,E2 9370.692} C_VEL
LIN {X 0,Y 310.086,Z 353.283,A -85,B 0,C 180,E1 9367.038,E2 9367.038} C_VEL
LIN {X 0,Y 308.229,Z 350.217,A -85,B 0,C 180,E1 9360.372,E2 9360.372} C_VEL
LIN {X 0,Y 308.543,Z 351.383,A -85,B 0,C 180,E1 9357.028,E2 9357.028} C_VEL
LIN {X 0,Y 310.417,Z 353.8,A -85,B 0,C 180,E1 9352.69,E2 9352.69} C_VEL
LIN {X 0,Y 313.235,Z 358.787,A -85,B 0,C 180,E1 9348.865,E2 9348.865} C_VEL
LIN {X 0,Y 316.054,Z 363.651,A -85,B 0,C 180,E1 9346.087,E2 9346.087} C_VEL
LIN {X 0,Y 319.911,Z 370.224,A -85,B 0,C 180,E1 9343.055,E2 9343.055} C_VEL
LIN {X 0,Y 324.562,Z 378.974,A -85,B 0,C 180,E1 9340.003,E2 9340.003} C_VEL
LIN {X 0,Y 326.998,Z 384.126,A -85,B 0,C 180,E1 9338.567,E2 9338.567} C_VEL
LIN {X 0,Y 329.243,Z 390.072,A -85,B 0,C 180,E1 9337.272,E2 9337.272} C_VEL
LIN {X 0,Y 317.46,Z 517.188,A -85,B 0,C 180,E1 9335.042,E2 9335.042} C_VEL
LIN {X 0,Y 314.091,Z 539.071,A -85,B 0,C 180,E1 9334.526,E2 9334.526} C_VEL
LIN {X 0,Y 309.086,Z 560.957,A -85,B 0,C 180,E1 9333.82,E2 9333.82} C_VEL
LIN {X 0,Y 303.929,Z 578.902,A -85,B 0,C 180,E1 9333.054,E2 9333.054} C_VEL
LIN {X 0,Y 298.408,Z 595.148,A -85,B 0,C 180,E1 9332.187,E2 9332.187} C_VEL
LIN {X 0,Y 292.203,Z 611.007,A -85,B 0,C 180,E1 9331.15,E2 9331.15} C_VEL
LIN {X 0,Y 285.35,Z 626.444,A -85,B 0,C 180,E1 9329.927,E2 9329.927} C_VEL
LIN {X 0,Y 277.922,Z 641.42,A -85,B 0,C 180,E1 9328.49,E2 9328.49} C_VEL
LIN {X 0,Y 269.262,Z 657.145,A -85,B 0,C 180,E1 9326.659,E2 9326.659} C_VEL
LIN {X 0,Y 262.112,Z 668.947,A -85,B 0,C 180,E1 9324.998,E2 9324.998} C_VEL
LIN {X 0,Y 257.911,Z 674.655,A -85,B 0,C 180,E1 9324.282,E2 9324.282} C_VEL
LIN {X 0,Y 244.653,Z 688.435,A -85,B 0,C 180,E1 9322.838,E2 9322.838} C_VEL
LIN {X 0,Y 240.289,Z 693.538,A -85,B 0,C 180,E1 9321.941,E2 9321.941} C_VEL
LIN {X 0,Y 228.412,Z 708.69,A -85,B 0,C 180,E1 9318.081,E2 9318.081} C_VEL
LIN {X 0,Y 219.395,Z 719.447,A -85,B 0,C 180,E1 9314.568,E2 9314.568} C_VEL
LIN {X 0,Y 211.742,Z 728.241,A -85,B 0,C 180,E1 9311.018,E2 9311.018} C_VEL
LIN {X 0,Y 204.51,Z 736.372,A -85,B 0,C 180,E1 9306.962,E2 9306.962} C_VEL
LIN {X 0,Y 198.318,Z 743.323,A -85,B 0,C 180,E1 9302.643,E2 9302.643} C_VEL
LIN {X 0,Y 192.952,Z 749.513,A -85,B 0,C 180,E1 9297.796,E2 9297.796} C_VEL
LIN {X 0,Y 188.682,Z 754.819,A -85,B 0,C 180,E1 9292.427,E2 9292.427} C_VEL
LIN {X 0,Y 185.32,Z 759.864,A -85,B 0,C 180,E1 9285.328,E2 9285.328} C_VEL
LIN {X 0,Y 184.116,Z 762.571,A -85,B 0,C 180,E1 9279.06,E2 9279.06} C_VEL
LIN {X 0,Y 183.962,Z 763.806,A -85,B 0,C 180,E1 9273.739,E2 9273.739} C_VEL
LIN {X 0,Y 183.995,Z 764.046,A -85,B 0,C 180,E1 9268.755,E2 9268.755} C_VEL
LIN {X 0,Y 183.982,Z 763.289,A -85,B 0,C 180,E1 9263.447,E2 9263.447} C_VEL
LIN {X 0,Y 184.541,Z 761.358,A -85,B 0,C 180,E1 9257.802,E2 9257.802} C_VEL
LIN {X 0,Y 186.233,Z 758.273,A -85,B 0,C 180,E1 9252.182,E2 9252.182} C_VEL
LIN {X 0,Y 189.111,Z 754.24,A -85,B 0,C 180,E1 9246.926,E2 9246.926} C_VEL
LIN {X 0,Y 193.231,Z 749.179,A -85,B 0,C 180,E1 9241.912,E2 9241.912} C_VEL
LIN {X 0,Y 198.674,Z 742.922,A -85,B 0,C 180,E1 9237.08,E2 9237.08} C_VEL
LIN {X 0,Y 205.359,Z 735.434,A -85,B 0,C 180,E1 9232.516,E2 9232.516} C_VEL
LIN {X 0,Y 214.716,Z 724.988,A -85,B 0,C 180,E1 9227.535,E2 9227.535} C_VEL
LIN {X 0,Y 224.931,Z 712.899,A -85,B 0,C 180,E1 9223.203,E2 9223.203} C_VEL
LIN {X 0,Y 233.827,Z 701.885,A -85,B 0,C 180,E1 9220.063,E2 9220.063} C_VEL
LIN {X 0,Y 242.72,Z 690.198,A -85,B 0,C 180,E1 9217.349,E2 9217.349} C_VEL
LIN {X 0,Y 251.783,Z 677.42,A -85,B 0,C 180,E1 9214.92,E2 9214.92} C_VEL
LIN {X 0,Y 260.913,Z 663.455,A -85,B 0,C 180,E1 9212.747,E2 9212.747} C_VEL
LIN {X 0,Y 271.912,Z 644.796,A -85,B 0,C 180,E1 9210.436,E2 9210.436} C_VEL
LIN {X 0,Y 280.623,Z 627.878,A -85,B 0,C 180,E1 9208.788,E2 9208.788} C_VEL
LIN {X 0,Y 287.617,Z 612.67,A -85,B 0,C 180,E1 9207.579,E2 9207.579} C_VEL
LIN {X 0,Y 293.943,Z 597.095,A -85,B 0,C 180,E1 9206.554,E2 9206.554} C_VEL
LIN {X 0,Y 299.563,Z 581.212,A -85,B 0,C 180,E1 9205.698,E2 9205.698} C_VEL
LIN {X 0,Y 304.436,Z 565.082,A -85,B 0,C 180,E1 9204.992,E2 9204.992} C_VEL
LIN {X 0,Y 308.781,Z 547.752,A -85,B 0,C 180,E1 9204.396,E2 9204.396} C_VEL
LIN {X 0,Y 312.249,Z 530.064,A -85,B 0,C 180,E1 9203.922,E2 9203.922} C_VEL
LIN {X 0,Y 314.99,Z 509.891,A -85,B 0,C 180,E1 9203.492,E2 9203.492} C_VEL
LIN {X 0,Y 325.812,Z 393.755,A -85,B 0,C 180,E1 9201.471,E2 9201.471} C_VEL
LIN {X 0,Y 322.96,Z 386.915,A -85,B 0,C 180,E1 9199.723,E2 9199.723} C_VEL
LIN {X 0,Y 318.347,Z 377.955,A -85,B 0,C 180,E1 9196.608,E2 9196.608} C_VEL
LIN {X 0,Y 314.749,Z 371.563,A -85,B 0,C 180,E1 9193.69,E2 9193.69} C_VEL
LIN {X 0,Y 312.811,Z 368.169,A -85,B 0,C 180,E1 9191.805,E2 9191.805} C_VEL
LIN {X 0,Y 311.241,Z 365.297,A -85,B 0,C 180,E1 9189.99,E2 9189.99} C_VEL
LIN {X 0,Y 308.97,Z 361.136,A -85,B 0,C 180,E1 9186.504,E2 9186.504} C_VEL
LIN {X 0,Y 307.251,Z 358.174,A -85,B 0,C 180,E1 9180,E2 9180} C_VEL
LIN {X 0,Y 307.624,Z 359.504,A -85,B 0,C 180,E1 9176.459,E2 9176.459} C_VEL
LIN {X 0,Y 309.255,Z 361.612,A -85,B 0,C 180,E1 9172.663,E2 9172.663} C_VEL
LIN {X 0,Y 311.975,Z 366.6,A -85,B 0,C 180,E1 9168.819,E2 9168.819} C_VEL
LIN {X 0,Y 314.624,Z 371.33,A -85,B 0,C 180,E1 9166.117,E2 9166.117} C_VEL
LIN {X 0,Y 318.083,Z 377.428,A -85,B 0,C 180,E1 9163.284,E2 9163.284} C_VEL
LIN {X 0,Y 322.506,Z 386.079,A -85,B 0,C 180,E1 9160.249,E2 9160.249} C_VEL
LIN {X 0,Y 327.229,Z 395.635,A -85,B 0,C 180,E1 9157.498,E2 9157.498} C_VEL
LIN {X 0,Y 336.757,Z 413.871,A -85,B 0,C 180,E1 9152.981,E2 9152.981} C_VEL
LIN {X 0,Y 348.484,Z 429.929,A -85,B 0,C 180,E1 9148.76,E2 9148.76} C_VEL
LIN {X 0,Y 361.602,Z 443.997,A -85,B 0,C 180,E1 9144.986,E2 9144.986} C_VEL
LIN {X 0,Y 388.136,Z 466.146,A -85,B 0,C 180,E1 9139.082,E2 9139.082} C_VEL
LIN {X 0,Y 398.388,Z 474.027,A -85,B 0,C 180,E1 9136.996,E2 9136.996} C_VEL
LIN {X 0,Y 408.778,Z 482.069,A -85,B 0,C 180,E1 9134.718,E2 9134.718} C_VEL
LIN {X 0,Y 418.074,Z 489.506,A -85,B 0,C 180,E1 9132.453,E2 9132.453} C_VEL
LIN {X 0,Y 426.043,Z 495.822,A -85,B 0,C 180,E1 9130.346,E2 9130.346} C_VEL
LIN {X 0,Y 434.394,Z 502.376,A -85,B 0,C 180,E1 9127.966,E2 9127.966} C_VEL
LIN {X 0,Y 442.894,Z 509.34,A -85,B 0,C 180,E1 9125.412,E2 9125.412} C_VEL
LIN {X 0,Y 450.322,Z 515.344,A -85,B 0,C 180,E1 9123.061,E2 9123.061} C_VEL
LIN {X 0,Y 457.951,Z 520.923,A -85,B 0,C 180,E1 9120.531,E2 9120.531} C_VEL
LIN {X 0,Y 464.963,Z 526.638,A -85,B 0,C 180,E1 9118.021,E2 9118.021} C_VEL
LIN {X 0,Y 471.442,Z 531.242,A -85,B 0,C 180,E1 9115.554,E2 9115.554} C_VEL
LIN {X 0,Y 477.281,Z 535.946,A -85,B 0,C 180,E1 9113.118,E2 9113.118} C_VEL
LIN {X 0,Y 482.859,Z 539.501,A -85,B 0,C 180,E1 9110.609,E2 9110.609} C_VEL
LIN {X 0,Y 487.544,Z 543.508,A -85,B 0,C 180,E1 9108.161,E2 9108.161} C_VEL
LIN {X 0,Y 492.028,Z 546.723,A -85,B 0,C 180,E1 9105.558,E2 9105.558} C_VEL
LIN {X 0,Y 495.853,Z 548.807,A -85,B 0,C 180,E1 9103.051,E2 9103.051} C_VEL
LIN {X 0,Y 497.728,Z 549.979,A -85,B 0,C 180,E1 9101.587,E2 9101.587} C_VEL
LIN {X 0,Y 500.259,Z 552.472,A -85,B 0,C 180,E1 9099.111,E2 9099.111} C_VEL
LIN {X 0,Y 502.245,Z 554.174,A -85,B 0,C 180,E1 9096.745,E2 9096.745} C_VEL
LIN {X 0,Y 503.627,Z 555.237,A -85,B 0,C 180,E1 9094.212,E2 9094.212} C_VEL
LIN {X 0,Y 504.484,Z 555.772,A -85,B 0,C 180,E1 9091.703,E2 9091.703} C_VEL
LIN {X 0,Y 504.531,Z 555.806,A -85,B 0,C 180,E1 9089.205,E2 9089.205} C_VEL
LIN {X 0,Y 504.062,Z 555.504,A -85,B 0,C 180,E1 9086.703,E2 9086.703} C_VEL
LIN {X 0,Y 502.783,Z 554.611,A -85,B 0,C 180,E1 9084.18,E2 9084.18} C_VEL
LIN {X 0,Y 501.078,Z 553.206,A -85,B 0,C 180,E1 9081.741,E2 9081.741} C_VEL
LIN {X 0,Y 498.608,Z 550.954,A -85,B 0,C 180,E1 9079.253,E2 9079.253} C_VEL
LIN {X 0,Y 496.614,Z 549.172,A -85,B 0,C 180,E1 9077.557,E2 9077.557} C_VEL
LIN {X 0,Y 492.846,Z 547.208,A -85,B 0,C 180,E1 9074.951,E2 9074.951} C_VEL
LIN {X 0,Y 488.787,Z 544.447,A -85,B 0,C 180,E1 9072.502,E2 9072.502} C_VEL
LIN {X 0,Y 484.083,Z 540.542,A -85,B 0,C 180,E1 9070.022,E2 9070.022} C_VEL
LIN {X 0,Y 479.422,Z 537.416,A -85,B 0,C 180,E1 9067.822,E2 9067.822} C_VEL
LIN {X 0,Y 473.869,Z 533.3,A -85,B 0,C 180,E1 9065.428,E2 9065.428} C_VEL
LIN {X 0,Y 468.963,Z 529.392,A -85,B 0,C 180,E1 9063.473,E2 9063.473} C_VEL
LIN {X 0,Y 462.37,Z 524.648,A -85,B 0,C 180,E1 9061.031,E2 9061.031} C_VEL
LIN {X 0,Y 455.731,Z 519.411,A -85,B 0,C 180,E1 9058.713,E2 9058.713} C_VEL
LIN {X 0,Y 448.239,Z 513.611,A -85,B 0,C 180,E1 9056.264,E2 9056.264} C_VEL
LIN {X 0,Y 440.596,Z 507.578,A -85,B 0,C 180,E1 9053.892,E2 9053.892} C_VEL
LIN {X 0,Y 431.595,Z 500.309,A -85,B 0,C 180,E1 9051.222,E2 9051.222} C_VEL
LIN {X 0,Y 423.757,Z 493.859,A -85,B 0,C 180,E1 9049.032,E2 9049.032} C_VEL
LIN {X 0,Y 415.199,Z 487.16,A -85,B 0,C 180,E1 9046.81,E2 9046.81} C_VEL
LIN {X 0,Y 405.496,Z 479.592,A -85,B 0,C 180,E1 9044.55,E2 9044.55} C_VEL
LIN {X 0,Y 395.669,Z 472.007,A -85,B 0,C 180,E1 9042.434,E2 9042.434} C_VEL
LIN {X 0,Y 381.747,Z 461.366,A -85,B 0,C 180,E1 9039.65,E2 9039.65} C_VEL
LIN {X 0,Y 355.413,Z 437.827,A -85,B 0,C 180,E1 9033.332,E2 9033.332} C_VEL
LIN {X 0,Y 341.579,Z 421.004,A -85,B 0,C 180,E1 9028.881,E2 9028.881} C_VEL
LIN {X 0,Y 331.403,Z 404.469,A -85,B 0,C 180,E1 9024.653,E2 9024.653} C_VEL
LIN {X 0,Y 324.77,Z 390.501,A -85,B 0,C 180,E1 9021.113,E2 9021.113} C_VEL
LIN {X 0,Y 319.461,Z 380.067,A -85,B 0,C 180,E1 9017.721,E2 9017.721} C_VEL
LIN {X 0,Y 315.641,Z 373.078,A -85,B 0,C 180,E1 9014.774,E2 9014.774} C_VEL
LIN {X 0,Y 312.96,Z 368.415,A -85,B 0,C 180,E1 9012.267,E2 9012.267} C_VEL
LIN {X 0,Y 311.141,Z 365.183,A -85,B 0,C 180,E1 9010.18,E2 9010.18} C_VEL
LIN {X 0,Y 309.007,Z 361.168,A -85,B 0,C 180,E1 9006.876,E2 9006.876} C_VEL
LIN {X 0,Y 307.254,Z 358.159,A -85,B 0,C 180,E1 9000.373,E2 9000.373} C_VEL
LIN {X 0,Y 307.564,Z 359.366,A -85,B 0,C 180,E1 8997.018,E2 8997.018} C_VEL
LIN {X 0,Y 309.288,Z 361.673,A -85,B 0,C 180,E1 8992.911,E2 8992.911} C_VEL
LIN {X 0,Y 311.921,Z 366.49,A -85,B 0,C 180,E1 8989.191,E2 8989.191} C_VEL
LIN {X 0,Y 314.555,Z 371.199,A -85,B 0,C 180,E1 8986.489,E2 8986.489} C_VEL
LIN {X 0,Y 318.231,Z 377.72,A -85,B 0,C 180,E1 8983.48,E2 8983.48} C_VEL
LIN {X 0,Y 322.683,Z 386.388,A -85,B 0,C 180,E1 8980.448,E2 8980.448} C_VEL
LIN {X 0,Y 324.889,Z 391.427,A -85,B 0,C 180,E1 8979.083,E2 8979.083} C_VEL
LIN {X 0,Y 325.832,Z 394.11,A -85,B 0,C 180,E1 8978.5,E2 8978.5} C_VEL
LIN {X 0,Y 314.154,Z 517.073,A -85,B 0,C 180,E1 8976.368,E2 8976.368} C_VEL
LIN {X 0,Y 310.638,Z 539.412,A -85,B 0,C 180,E1 8975.848,E2 8975.848} C_VEL
LIN {X 0,Y 305.541,Z 561.103,A -85,B 0,C 180,E1 8975.159,E2 8975.159} C_VEL
LIN {X 0,Y 300.373,Z 578.726,A -85,B 0,C 180,E1 8974.421,E2 8974.421} C_VEL
LIN {X 0,Y 294.738,Z 594.972,A -85,B 0,C 180,E1 8973.571,E2 8973.571} C_VEL
LIN {X 0,Y 288.4,Z 610.831,A -85,B 0,C 180,E1 8972.553,E2 8972.553} C_VEL
LIN {X 0,Y 281.392,Z 626.268,A -85,B 0,C 180,E1 8971.35,E2 8971.35} C_VEL
LIN {X 0,Y 273.783,Z 641.243,A -85,B 0,C 180,E1 8969.932,E2 8969.932} C_VEL
LIN {X 0,Y 264.897,Z 656.968,A -85,B 0,C 180,E1 8968.122,E2 8968.122} C_VEL
LIN {X 0,Y 253.167,Z 675.424,A -85,B 0,C 180,E1 8965.423,E2 8965.423} C_VEL
LIN {X 0,Y 243.47,Z 689.181,A -85,B 0,C 180,E1 8962.864,E2 8962.864} C_VEL
LIN {X 0,Y 240.289,Z 693.538,A -85,B 0,C 180,E1 8961.941,E2 8961.941} C_VEL
LIN {X 0,Y 235.886,Z 698.555,A -85,B 0,C 180,E1 8960.981,E2 8960.981} C_VEL
LIN {X 0,Y 222.037,Z 710.463,A -85,B 0,C 180,E1 8958.86,E2 8958.86} C_VEL
LIN {X 0,Y 217.611,Z 714.889,A -85,B 0,C 180,E1 8957.668,E2 8957.668} C_VEL
LIN {X 0,Y 206.667,Z 726.979,A -85,B 0,C 180,E1 8953.007,E2 8953.007} C_VEL
LIN {X 0,Y 198.48,Z 735.724,A -85,B 0,C 180,E1 8948.652,E2 8948.652} C_VEL
LIN {X 0,Y 191.86,Z 742.744,A -85,B 0,C 180,E1 8944.248,E2 8944.248} C_VEL
LIN {X 0,Y 186.061,Z 749,A -85,B 0,C 180,E1 8939.273,E2 8939.273} C_VEL
LIN {X 0,Y 181.604,Z 754.099,A -85,B 0,C 180,E1 8934.04,E2 8934.04} C_VEL
LIN {X 0,Y 178.364,Z 758.305,A -85,B 0,C 180,E1 8928.294,E2 8928.294} C_VEL
LIN {X 0,Y 176.347,Z 761.923,A -85,B 0,C 180,E1 8921.114,E2 8921.114} C_VEL
LIN {X 0,Y 175.958,Z 763.6,A -85,B 0,C 180,E1 8914.236,E2 8914.236} C_VEL
LIN {X 0,Y 175.999,Z 763.901,A -85,B 0,C 180,E1 8909.024,E2 8909.024} C_VEL
LIN {X 0,Y 175.99,Z 763.113,A -85,B 0,C 180,E1 8903.149,E2 8903.149} C_VEL
LIN {X 0,Y 176.636,Z 761.181,A -85,B 0,C 180,E1 8897.248,E2 8897.248} C_VEL
LIN {X 0,Y 178.506,Z 758.095,A -85,B 0,C 180,E1 8891.383,E2 8891.383} C_VEL
LIN {X 0,Y 181.604,Z 754.098,A -85,B 0,C 180,E1 8885.96,E2 8885.96} C_VEL
LIN {X 0,Y 186.06,Z 749,A -85,B 0,C 180,E1 8880.727,E2 8880.727} C_VEL
LIN {X 0,Y 191.86,Z 742.744,A -85,B 0,C 180,E1 8875.752,E2 8875.752} C_VEL
LIN {X 0,Y 198.93,Z 735.255,A -85,B 0,C 180,E1 8871.082,E2 8871.082} C_VEL
LIN {X 0,Y 208.76,Z 724.809,A -85,B 0,C 180,E1 8866.02,E2 8866.02} C_VEL
LIN {X 0,Y 219.423,Z 712.721,A -85,B 0,C 180,E1 8861.649,E2 8861.649} C_VEL
LIN {X 0,Y 228.665,Z 701.707,A -85,B 0,C 180,E1 8858.5,E2 8858.5} C_VEL
LIN {X 0,Y 237.872,Z 690.02,A -85,B 0,C 180,E1 8855.79,E2 8855.79} C_VEL
LIN {X 0,Y 246.867,Z 677.742,A -85,B 0,C 180,E1 8853.462,E2 8853.462} C_VEL
LIN {X 0,Y 255.881,Z 664.399,A -85,B 0,C 180,E1 8851.383,E2 8851.383} C_VEL
LIN {X 0,Y 265.995,Z 647.973,A -85,B 0,C 180,E1 8849.31,E2 8849.31} C_VEL
LIN {X 0,Y 276.433,Z 628.507,A -85,B 0,C 180,E1 8847.392,E2 8847.392} C_VEL
LIN {X 0,Y 283.975,Z 612.494,A -85,B 0,C 180,E1 8846.137,E2 8846.137} C_VEL
LIN {X 0,Y 290.433,Z 596.919,A -85,B 0,C 180,E1 8845.133,E2 8845.133} C_VEL
LIN {X 0,Y 296.166,Z 581.036,A -85,B 0,C 180,E1 8844.297,E2 8844.297} C_VEL
LIN {X 0,Y 301.133,Z 564.907,A -85,B 0,C 180,E1 8843.607,E2 8843.607} C_VEL
LIN {X 0,Y 305.556,Z 547.576,A -85,B 0,C 180,E1 8843.026,E2 8843.026} C_VEL
LIN {X 0,Y 309.11,Z 529.743,A -85,B 0,C 180,E1 8842.56,E2 8842.56} C_VEL
LIN {X 0,Y 311.967,Z 508.997,A -85,B 0,C 180,E1 8842.127,E2 8842.127} C_VEL
LIN {X 0,Y 322.542,Z 397.998,A -85,B 0,C 180,E1 8840.222,E2 8840.222} C_VEL
LIN {X 0,Y 320.557,Z 393.268,A -85,B 0,C 180,E1 8838.929,E2 8838.929} C_VEL
LIN {X 0,Y 316.29,Z 384.631,A -85,B 0,C 180,E1 8835.87,E2 8835.87} C_VEL
LIN {X 0,Y 312.266,Z 377.113,A -85,B 0,C 180,E1 8832.295,E2 8832.295} C_VEL
LIN {X 0,Y 309.962,Z 373,A -85,B 0,C 180,E1 8829.657,E2 8829.657} C_VEL
LIN {X 0,Y 307.893,Z 369.02,A -85,B 0,C 180,E1 8826.339,E2 8826.339} C_VEL
LIN {X 0,Y 306.276,Z 366.115,A -85,B 0,C 180,E1 8820,E2 8820} C_VEL
LIN {X 0,Y 306.695,Z 367.578,A -85,B 0,C 180,E1 8816.261,E2 8816.261} C_VEL
LIN {X 0,Y 308.162,Z 369.572,A -85,B 0,C 180,E1 8812.824,E2 8812.824} C_VEL
LIN {X 0,Y 310.67,Z 374.303,A -85,B 0,C 180,E1 8809.147,E2 8809.147} C_VEL
LIN {X 0,Y 313.233,Z 379.059,A -85,B 0,C 180,E1 8806.431,E2 8806.431} C_VEL
LIN {X 0,Y 316.538,Z 385.161,A -85,B 0,C 180,E1 8803.625,E2 8803.625} C_VEL
LIN {X 0,Y 321.194,Z 394.536,A -85,B 0,C 180,E1 8800.354,E2 8800.354} C_VEL
LIN {X 0,Y 325.606,Z 404.097,A -85,B 0,C 180,E1 8797.713,E2 8797.713} C_VEL
LIN {X 0,Y 335.254,Z 422.448,A -85,B 0,C 180,E1 8793.09,E2 8793.09} C_VEL
LIN {X 0,Y 348.68,Z 440.464,A -85,B 0,C 180,E1 8788.298,E2 8788.298} C_VEL
LIN {X 0,Y 369.349,Z 460.645,A -85,B 0,C 180,E1 8782.767,E2 8782.767} C_VEL
LIN {X 0,Y 393.283,Z 479.503,A -85,B 0,C 180,E1 8777.791,E2 8777.791} C_VEL
LIN {X 0,Y 404.023,Z 487.735,A -85,B 0,C 180,E1 8775.493,E2 8775.493} C_VEL
LIN {X 0,Y 412.459,Z 494.257,A -85,B 0,C 180,E1 8773.544,E2 8773.544} C_VEL
LIN {X 0,Y 422.212,Z 501.796,A -85,B 0,C 180,E1 8771.089,E2 8771.089} C_VEL
LIN {X 0,Y 430.647,Z 508.612,A -85,B 0,C 180,E1 8768.727,E2 8768.727} C_VEL
LIN {X 0,Y 440.308,Z 516.374,A -85,B 0,C 180,E1 8765.86,E2 8765.86} C_VEL
LIN {X 0,Y 448.076,Z 522.552,A -85,B 0,C 180,E1 8763.443,E2 8763.443} C_VEL
LIN {X 0,Y 455.525,Z 528.066,A -85,B 0,C 180,E1 8761.001,E2 8761.001} C_VEL
LIN {X 0,Y 462.99,Z 534.028,A -85,B 0,C 180,E1 8758.363,E2 8758.363} C_VEL
LIN {X 0,Y 470,Z 539,A -85,B 0,C 180,E1 8755.718,E2 8755.718} C_VEL
LIN {X 0,Y 475.947,Z 543.746,A -85,B 0,C 180,E1 8753.26,E2 8753.26} C_VEL
LIN {X 0,Y 481.404,Z 547.246,A -85,B 0,C 180,E1 8750.801,E2 8750.801} C_VEL
LIN {X 0,Y 486.386,Z 551.408,A -85,B 0,C 180,E1 8748.238,E2 8748.238} C_VEL
LIN {X 0,Y 490.779,Z 554.532,A -85,B 0,C 180,E1 8745.72,E2 8745.72} C_VEL
LIN {X 0,Y 494.63,Z 556.653,A -85,B 0,C 180,E1 8743.203,E2 8743.203} C_VEL
LIN {X 0,Y 496.699,Z 557.948,A -85,B 0,C 180,E1 8741.612,E2 8741.612} C_VEL
LIN {X 0,Y 499.262,Z 560.432,A -85,B 0,C 180,E1 8739.122,E2 8739.122} C_VEL
LIN {X 0,Y 501.251,Z 562.116,A -85,B 0,C 180,E1 8736.758,E2 8736.758} C_VEL
LIN {X 0,Y 502.646,Z 563.179,A -85,B 0,C 180,E1 8734.22,E2 8734.22} C_VEL
LIN {X 0,Y 503.509,Z 563.712,A -85,B 0,C 180,E1 8731.707,E2 8731.707} C_VEL
LIN {X 0,Y 503.555,Z 563.746,A -85,B 0,C 180,E1 8729.204,E2 8729.204} C_VEL
LIN {X 0,Y 503.085,Z 563.444,A -85,B 0,C 180,E1 8726.696,E2 8726.696} C_VEL
LIN {X 0,Y 501.797,Z 562.552,A -85,B 0,C 180,E1 8724.168,E2 8724.168} C_VEL
LIN {X 0,Y 500.082,Z 561.156,A -85,B 0,C 180,E1 8721.724,E2 8721.724} C_VEL
LIN {X 0,Y 497.594,Z 558.913,A -85,B 0,C 180,E1 8719.231,E2 8719.231} C_VEL
LIN {X 0,Y 495.442,Z 557.038,A -85,B 0,C 180,E1 8717.412,E2 8717.412} C_VEL
LIN {X 0,Y 491.584,Z 555.023,A -85,B 0,C 180,E1 8714.79,E2 8714.79} C_VEL
LIN {X 0,Y 487.476,Z 552.218,A -85,B 0,C 180,E1 8712.33,E2 8712.33} C_VEL
LIN {X 0,Y 482.821,Z 548.376,A -85,B 0,C 180,E1 8709.896,E2 8709.896} C_VEL
LIN {X 0,Y 477.754,Z 545.013,A -85,B 0,C 180,E1 8707.549,E2 8707.549} C_VEL
LIN {X 0,Y 472.138,Z 540.813,A -85,B 0,C 180,E1 8705.145,E2 8705.145} C_VEL
LIN {X 0,Y 467.332,Z 537.046,A -85,B 0,C 180,E1 8703.253,E2 8703.253} C_VEL
LIN {X 0,Y 460.542,Z 532.16,A -85,B 0,C 180,E1 8700.762,E2 8700.762} C_VEL
LIN {X 0,Y 453.934,Z 526.999,A -85,B 0,C 180,E1 8698.48,E2 8698.48} C_VEL
LIN {X 0,Y 446.284,Z 521.084,A -85,B 0,C 180,E1 8695.994,E2 8695.994} C_VEL
LIN {X 0,Y 437.348,Z 514.05,A -85,B 0,C 180,E1 8693.247,E2 8693.247} C_VEL
LIN {X 0,Y 428.766,Z 507.187,A -85,B 0,C 180,E1 8690.736,E2 8690.736} C_VEL
LIN {X 0,Y 419.878,Z 499.961,A -85,B 0,C 180,E1 8688.294,E2 8688.294} C_VEL
LIN {X 0,Y 411.538,Z 493.509,A -85,B 0,C 180,E1 8686.238,E2 8686.238} C_VEL
LIN {X 0,Y 402.044,Z 486.183,A -85,B 0,C 180,E1 8684.057,E2 8684.057} C_VEL
LIN {X 0,Y 390.882,Z 477.719,A -85,B 0,C 180,E1 8681.738,E2 8681.738} C_VEL
LIN {X 0,Y 365.382,Z 457.027,A -85,B 0,C 180,E1 8676.284,E2 8676.284} C_VEL
LIN {X 0,Y 348.331,Z 440.052,A -85,B 0,C 180,E1 8671.592,E2 8671.592} C_VEL
LIN {X 0,Y 334.967,Z 421.992,A -85,B 0,C 180,E1 8666.791,E2 8666.791} C_VEL
LIN {X 0,Y 325.382,Z 403.584,A -85,B 0,C 180,E1 8662.161,E2 8662.161} C_VEL
LIN {X 0,Y 320.922,Z 394.018,A -85,B 0,C 180,E1 8659.474,E2 8659.474} C_VEL
LIN {X 0,Y 316.482,Z 385.043,A -85,B 0,C 180,E1 8656.331,E2 8656.331} C_VEL
LIN {X 0,Y 313.139,Z 378.875,A -85,B 0,C 180,E1 8653.479,E2 8653.479} C_VEL
LIN {X 0,Y 310.165,Z 373.265,A -85,B 0,C 180,E1 8650.213,E2 8650.213} C_VEL
LIN {X 0,Y 307.827,Z 368.969,A -85,B 0,C 180,E1 8646.528,E2 8646.528} C_VEL
LIN {X 0,Y 306.276,Z 366.106,A -85,B 0,C 180,E1 8640.187,E2 8640.187} C_VEL
LIN {X 0,Y 307.181,Z 368.286,A -85,B 0,C 180,E1 8635.145,E2 8635.145} C_VEL
LIN {X 0,Y 308.178,Z 369.584,A -85,B 0,C 180,E1 8633.105,E2 8633.105} C_VEL
LIN {X 0,Y 310.617,Z 374.192,A -85,B 0,C 180,E1 8629.521,E2 8629.521} C_VEL
LIN {X 0,Y 313.164,Z 378.928,A -85,B 0,C 180,E1 8626.803,E2 8626.803} C_VEL
LIN {X 0,Y 316.625,Z 385.33,A -85,B 0,C 180,E1 8623.865,E2 8623.865} C_VEL
LIN {X 0,Y 321.162,Z 394.452,A -85,B 0,C 180,E1 8620.683,E2 8620.683} C_VEL
LIN {X 0,Y 322.551,Z 398.39,A -85,B 0,C 180,E1 8619.749,E2 8619.749} C_VEL
LIN {X 0,Y 311.011,Z 517.033,A -85,B 0,C 180,E1 8617.718,E2 8617.718} C_VEL
LIN {X 0,Y 307.358,Z 539.704,A -85,B 0,C 180,E1 8617.2,E2 8617.2} C_VEL
LIN {X 0,Y 302.16,Z 561.274,A -85,B 0,C 180,E1 8616.526,E2 8616.526} C_VEL
LIN {X 0,Y 296.991,Z 578.55,A -85,B 0,C 180,E1 8615.819,E2 8615.819} C_VEL
LIN {X 0,Y 291.245,Z 594.796,A -85,B 0,C 180,E1 8614.989,E2 8614.989} C_VEL
LIN {X 0,Y 284.775,Z 610.654,A -85,B 0,C 180,E1 8613.992,E2 8613.992} C_VEL
LIN {X 0,Y 277.612,Z 626.091,A -85,B 0,C 180,E1 8612.812,E2 8612.812} C_VEL
LIN {X 0,Y 269.823,Z 641.066,A -85,B 0,C 180,E1 8611.418,E2 8611.418} C_VEL
LIN {X 0,Y 260.711,Z 656.791,A -85,B 0,C 180,E1 8609.634,E2 8609.634} C_VEL
LIN {X 0,Y 248.647,Z 675.246,A -85,B 0,C 180,E1 8606.964,E2 8606.964} C_VEL
LIN {X 0,Y 239.231,Z 688.241,A -85,B 0,C 180,E1 8604.578,E2 8604.578} C_VEL
LIN {X 0,Y 229.949,Z 700.125,A -85,B 0,C 180,E1 8601.9,E2 8601.9} C_VEL
LIN {X 0,Y 221.219,Z 710.616,A -85,B 0,C 180,E1 8599.001,E2 8599.001} C_VEL
LIN {X 0,Y 217.611,Z 714.889,A -85,B 0,C 180,E1 8597.668,E2 8597.668} C_VEL
LIN {X 0,Y 213.216,Z 719.164,A -85,B 0,C 180,E1 8596.4,E2 8596.4} C_VEL
LIN {X 0,Y 199.404,Z 729.076,A -85,B 0,C 180,E1 8593.399,E2 8593.399} C_VEL
LIN {X 0,Y 195.154,Z 732.647,A -85,B 0,C 180,E1 8591.821,E2 8591.821} C_VEL
LIN {X 0,Y 185.939,Z 741.794,A -85,B 0,C 180,E1 8586.232,E2 8586.232} C_VEL
LIN {X 0,Y 179.632,Z 748.152,A -85,B 0,C 180,E1 8581.171,E2 8581.171} C_VEL
LIN {X 0,Y 174.677,Z 753.378,A -85,B 0,C 180,E1 8575.784,E2 8575.784} C_VEL
LIN {X 0,Y 171.135,Z 757.498,A -85,B 0,C 180,E1 8570.162,E2 8570.162} C_VEL
LIN {X 0,Y 168.991,Z 760.556,A -85,B 0,C 180,E1 8564.387,E2 8564.387} C_VEL
LIN {X 0,Y 168.075,Z 762.578,A -85,B 0,C 180,E1 8558.552,E2 8558.552} C_VEL
LIN {X 0,Y 167.967,Z 763.517,A -85,B 0,C 180,E1 8553.412,E2 8553.412} C_VEL
LIN {X 0,Y 167.996,Z 763.697,A -85,B 0,C 180,E1 8548.636,E2 8548.636} C_VEL
LIN {X 0,Y 168,Z 762.937,A -85,B 0,C 180,E1 8542.821,E2 8542.821} C_VEL
LIN {X 0,Y 168.746,Z 761.004,A -85,B 0,C 180,E1 8536.641,E2 8536.641} C_VEL
LIN {X 0,Y 170.849,Z 757.869,A -85,B 0,C 180,E1 8530.434,E2 8530.434} C_VEL
LIN {X 0,Y 174.186,Z 753.92,A -85,B 0,C 180,E1 8524.867,E2 8524.867} C_VEL
LIN {X 0,Y 178.976,Z 748.821,A -85,B 0,C 180,E1 8519.448,E2 8519.448} C_VEL
LIN {X 0,Y 185.155,Z 742.565,A -85,B 0,C 180,E1 8514.327,E2 8514.327} C_VEL
LIN {X 0,Y 192.634,Z 735.076,A -85,B 0,C 180,E1 8509.554,E2 8509.554} C_VEL
LIN {X 0,Y 203.107,Z 724.478,A -85,B 0,C 180,E1 8504.352,E2 8504.352} C_VEL
LIN {X 0,Y 214.087,Z 712.542,A -85,B 0,C 180,E1 8500.017,E2 8500.017} C_VEL
LIN {X 0,Y 223.684,Z 701.529,A -85,B 0,C 180,E1 8496.866,E2 8496.866} C_VEL
LIN {X 0,Y 233.207,Z 689.842,A -85,B 0,C 180,E1 8494.169,E2 8494.169} C_VEL
LIN {X 0,Y 242.516,Z 677.52,A -85,B 0,C 180,E1 8491.853,E2 8491.853} C_VEL
LIN {X 0,Y 251.753,Z 664.222,A -85,B 0,C 180,E1 8489.808,E2 8489.808} C_VEL
LIN {X 0,Y 262.129,Z 647.796,A -85,B 0,C 180,E1 8487.768,E2 8487.768} C_VEL
LIN {X 0,Y 272.813,Z 628.331,A -85,B 0,C 180,E1 8485.887,E2 8485.887} C_VEL
LIN {X 0,Y 280.694,Z 611.92,A -85,B 0,C 180,E1 8484.632,E2 8484.632} C_VEL
LIN {X 0,Y 287.106,Z 596.743,A -85,B 0,C 180,E1 8483.679,E2 8483.679} C_VEL
LIN {X 0,Y 292.951,Z 580.861,A -85,B 0,C 180,E1 8482.864,E2 8482.864} C_VEL
LIN {X 0,Y 298.01,Z 564.731,A -85,B 0,C 180,E1 8482.193,E2 8482.193} C_VEL
LIN {X 0,Y 302.509,Z 547.401,A -85,B 0,C 180,E1 8481.628,E2 8481.628} C_VEL
LIN {X 0,Y 306.108,Z 529.654,A -85,B 0,C 180,E1 8481.176,E2 8481.176} C_VEL
LIN {X 0,Y 308.985,Z 509.232,A -85,B 0,C 180,E1 8480.757,E2 8480.757} C_VEL
LIN {X 0,Y 319.436,Z 402.29,A -85,B 0,C 180,E1 8478.956,E2 8478.956} C_VEL
LIN {X 0,Y 315.594,Z 394.074,A -85,B 0,C 180,E1 8476.189,E2 8476.189} C_VEL
LIN {X 0,Y 312.062,Z 387.186,A -85,B 0,C 180,E1 8473.15,E2 8473.15} C_VEL
LIN {X 0,Y 309.994,Z 383.261,A -85,B 0,C 180,E1 8470.971,E2 8470.971} C_VEL
LIN {X 0,Y 308.555,Z 380.507,A -85,B 0,C 180,E1 8469.137,E2 8469.137} C_VEL
LIN {X 0,Y 306.721,Z 376.819,A -85,B 0,C 180,E1 8465.988,E2 8465.988} C_VEL
LIN {X 0,Y 305.301,Z 374.047,A -85,B 0,C 180,E1 8459.812,E2 8459.812} C_VEL
LIN {X 0,Y 306.945,Z 377.127,A -85,B 0,C 180,E1 8453.265,E2 8453.265} C_VEL
LIN {X 0,Y 309.447,Z 382.161,A -85,B 0,C 180,E1 8449.387,E2 8449.387} C_VEL
LIN {X 0,Y 311.76,Z 386.606,A -85,B 0,C 180,E1 8446.837,E2 8446.837} C_VEL
LIN {X 0,Y 314.842,Z 392.537,A -85,B 0,C 180,E1 8444.103,E2 8444.103} C_VEL
LIN {X 0,Y 319.278,Z 401.835,A -85,B 0,C 180,E1 8440.85,E2 8440.85} C_VEL
LIN {X 0,Y 323.478,Z 411.339,A -85,B 0,C 180,E1 8438.227,E2 8438.227} C_VEL
LIN {X 0,Y 332.903,Z 429.632,A -85,B 0,C 180,E1 8433.559,E2 8433.559} C_VEL
LIN {X 0,Y 346.341,Z 447.889,A -85,B 0,C 180,E1 8428.642,E2 8428.642} C_VEL
LIN {X 0,Y 367.376,Z 468.505,A -85,B 0,C 180,E1 8422.925,E2 8422.925} C_VEL
LIN {X 0,Y 391.881,Z 487.748,A -85,B 0,C 180,E1 8417.802,E2 8417.802} C_VEL
LIN {X 0,Y 402.688,Z 495.966,A -85,B 0,C 180,E1 8415.506,E2 8415.506} C_VEL
LIN {X 0,Y 410.647,Z 502.092,A -85,B 0,C 180,E1 8413.683,E2 8413.683} C_VEL
LIN {X 0,Y 419.396,Z 508.735,A -85,B 0,C 180,E1 8411.506,E2 8411.506} C_VEL
LIN {X 0,Y 428.02,Z 515.685,A -85,B 0,C 180,E1 8409.142,E2 8409.142} C_VEL
LIN {X 0,Y 437.596,Z 523.303,A -85,B 0,C 180,E1 8406.346,E2 8406.346} C_VEL
LIN {X 0,Y 445.368,Z 529.426,A -85,B 0,C 180,E1 8403.946,E2 8403.946} C_VEL
LIN {X 0,Y 453.048,Z 535.205,A -85,B 0,C 180,E1 8401.458,E2 8401.458} C_VEL
LIN {X 0,Y 460.822,Z 541.282,A -85,B 0,C 180,E1 8398.765,E2 8398.765} C_VEL
LIN {X 0,Y 468.201,Z 546.441,A -85,B 0,C 180,E1 8396.028,E2 8396.028} C_VEL
LIN {X 0,Y 474.029,Z 551.161,A -85,B 0,C 180,E1 8393.623,E2 8393.623} C_VEL
LIN {X 0,Y 479.641,Z 554.813,A -85,B 0,C 180,E1 8391.137,E2 8391.137} C_VEL
LIN {X 0,Y 484.531,Z 558.741,A -85,B 0,C 180,E1 8388.7,E2 8388.7} C_VEL
LIN {X 0,Y 488.887,Z 561.927,A -85,B 0,C 180,E1 8386.27,E2 8386.27} C_VEL
LIN {X 0,Y 492.837,Z 564.221,A -85,B 0,C 180,E1 8383.73,E2 8383.73} C_VEL
LIN {X 0,Y 495.51,Z 565.763,A -85,B 0,C 180,E1 8381.758,E2 8381.758} C_VEL
LIN {X 0,Y 498.17,Z 568.299,A -85,B 0,C 180,E1 8379.239,E2 8379.239} C_VEL
LIN {X 0,Y 500.054,Z 569.929,A -85,B 0,C 180,E1 8377.005,E2 8377.005} C_VEL
LIN {X 0,Y 501.617,Z 571.081,A -85,B 0,C 180,E1 8374.344,E2 8374.344} C_VEL
LIN {X 0,Y 502.413,Z 571.592,A -85,B 0,C 180,E1 8372.053,E2 8372.053} C_VEL
LIN {X 0,Y 502.605,Z 571.69,A -85,B 0,C 180,E1 8369.43,E2 8369.43} C_VEL
LIN {X 0,Y 502.198,Z 571.445,A -85,B 0,C 180,E1 8367.147,E2 8367.147} C_VEL
LIN {X 0,Y 501.029,Z 570.64,A -85,B 0,C 180,E1 8364.504,E2 8364.504} C_VEL
LIN {X 0,Y 499.419,Z 569.433,A -85,B 0,C 180,E1 8362.176,E2 8362.176} C_VEL
LIN {X 0,Y 496.972,Z 567.237,A -85,B 0,C 180,E1 8359.569,E2 8359.569} C_VEL
LIN {X 0,Y 494.421,Z 564.971,A -85,B 0,C 180,E1 8357.386,E2 8357.386} C_VEL
LIN {X 0,Y 490.738,Z 563.073,A -85,B 0,C 180,E1 8354.884,E2 8354.884} C_VEL
LIN {X 0,Y 486.64,Z 560.343,A -85,B 0,C 180,E1 8352.422,E2 8352.422} C_VEL
LIN {X 0,Y 481.839,Z 556.47,A -85,B 0,C 180,E1 8349.916,E2 8349.916} C_VEL
LIN {X 0,Y 477.958,Z 553.782,A -85,B 0,C 180,E1 8348.072,E2 8348.072} C_VEL
LIN {X 0,Y 472.163,Z 549.75,A -85,B 0,C 180,E1 8345.589,E2 8345.589} C_VEL
LIN {X 0,Y 466.096,Z 544.95,A -85,B 0,C 180,E1 8343.18,E2 8343.18} C_VEL
LIN {X 0,Y 459.216,Z 540.064,A -85,B 0,C 180,E1 8340.67,E2 8340.67} C_VEL
LIN {X 0,Y 452.618,Z 534.913,A -85,B 0,C 180,E1 8338.401,E2 8338.401} C_VEL
LIN {X 0,Y 444.918,Z 529.049,A -85,B 0,C 180,E1 8335.91,E2 8335.91} C_VEL
LIN {X 0,Y 436.671,Z 522.585,A -85,B 0,C 180,E1 8333.377,E2 8333.377} C_VEL
LIN {X 0,Y 427.547,Z 515.331,A -85,B 0,C 180,E1 8330.724,E2 8330.724} C_VEL
LIN {X 0,Y 418.597,Z 508.102,A -85,B 0,C 180,E1 8328.285,E2 8328.285} C_VEL
LIN {X 0,Y 410.097,Z 501.648,A -85,B 0,C 180,E1 8326.184,E2 8326.184} C_VEL
LIN {X 0,Y 400.924,Z 494.614,A -85,B 0,C 180,E1 8324.092,E2 8324.092} C_VEL
LIN {X 0,Y 390.071,Z 486.443,A -85,B 0,C 180,E1 8321.845,E2 8321.845} C_VEL
LIN {X 0,Y 363.421,Z 464.939,A -85,B 0,C 180,E1 8316.12,E2 8316.12} C_VEL
LIN {X 0,Y 345.425,Z 446.793,A -85,B 0,C 180,E1 8311.063,E2 8311.063} C_VEL
LIN {X 0,Y 332.342,Z 428.721,A -85,B 0,C 180,E1 8306.201,E2 8306.201} C_VEL
LIN {X 0,Y 322.973,Z 410.151,A -85,B 0,C 180,E1 8301.475,E2 8301.475} C_VEL
LIN {X 0,Y 318.821,Z 400.903,A -85,B 0,C 180,E1 8298.846,E2 8298.846} C_VEL
LIN {X 0,Y 314.575,Z 391.949,A -85,B 0,C 180,E1 8295.675,E2 8295.675} C_VEL
LIN {X 0,Y 310.893,Z 384.769,A -85,B 0,C 180,E1 8292.255,E2 8292.255} C_VEL
LIN {X 0,Y 308.604,Z 380.589,A -85,B 0,C 180,E1 8289.511,E2 8289.511} C_VEL
LIN {X 0,Y 306.756,Z 376.853,A -85,B 0,C 180,E1 8286.363,E2 8286.363} C_VEL
LIN {X 0,Y 305.301,Z 374.046,A -85,B 0,C 180,E1 8280.188,E2 8280.188} C_VEL
LIN {X 0,Y 306.919,Z 377.003,A -85,B 0,C 180,E1 8273.64,E2 8273.64} C_VEL
LIN {X 0,Y 309.394,Z 382.05,A -85,B 0,C 180,E1 8269.761,E2 8269.761} C_VEL
LIN {X 0,Y 311.693,Z 386.474,A -85,B 0,C 180,E1 8267.212,E2 8267.212} C_VEL
LIN {X 0,Y 314.979,Z 392.819,A -85,B 0,C 180,E1 8264.299,E2 8264.299} C_VEL
LIN {X 0,Y 319.179,Z 401.623,A -85,B 0,C 180,E1 8261.223,E2 8261.223} C_VEL
LIN {X 0,Y 319.425,Z 402.685,A -85,B 0,C 180,E1 8261.023,E2 8261.023} C_VEL
LIN {X 0,Y 308.06,Z 516.866,A -85,B 0,C 180,E1 8259.098,E2 8259.098} C_VEL
LIN {X 0,Y 304.311,Z 539.676,A -85,B 0,C 180,E1 8258.588,E2 8258.588} C_VEL
LIN {X 0,Y 299.077,Z 561.018,A -85,B 0,C 180,E1 8257.939,E2 8257.939} C_VEL
LIN {X 0,Y 293.791,Z 578.375,A -85,B 0,C 180,E1 8257.249,E2 8257.249} C_VEL
LIN {X 0,Y 287.935,Z 594.62,A -85,B 0,C 180,E1 8256.441,E2 8256.441} C_VEL
LIN {X 0,Y 281.334,Z 610.478,A -85,B 0,C 180,E1 8255.467,E2 8255.467} C_VEL
LIN {X 0,Y 274.02,Z 625.915,A -85,B 0,C 180,E1 8254.312,E2 8254.312} C_VEL
LIN {X 0,Y 266.05,Z 640.89,A -85,B 0,C 180,E1 8252.947,E2 8252.947} C_VEL
LIN {X 0,Y 256.712,Z 656.614,A -85,B 0,C 180,E1 8251.193,E2 8251.193} C_VEL
LIN {X 0,Y 244.316,Z 675.069,A -85,B 0,C 180,E1 8248.561,E2 8248.561} C_VEL
LIN {X 0,Y 234.611,Z 688.063,A -85,B 0,C 180,E1 8246.197,E2 8246.197} C_VEL
LIN {X 0,Y 225.015,Z 699.946,A -85,B 0,C 180,E1 8243.532,E2 8243.532} C_VEL
LIN {X 0,Y 215.916,Z 710.481,A -85,B 0,C 180,E1 8240.621,E2 8240.621} C_VEL
LIN {X 0,Y 206.91,Z 720.327,A -85,B 0,C 180,E1 8237.26,E2 8237.26} C_VEL
LIN {X 0,Y 198.367,Z 729.248,A -85,B 0,C 180,E1 8233.46,E2 8233.46} C_VEL
LIN {X 0,Y 195.154,Z 732.647,A -85,B 0,C 180,E1 8231.821,E2 8231.821} C_VEL
LIN {X 0,Y 191.017,Z 736.069,A -85,B 0,C 180,E1 8230.153,E2 8230.153} C_VEL
LIN {X 0,Y 178.035,Z 743.892,A -85,B 0,C 180,E1 8226.029,E2 8226.029} C_VEL
LIN {X 0,Y 174.322,Z 746.487,A -85,B 0,C 180,E1 8223.976,E2 8223.976} C_VEL
LIN {X 0,Y 167.914,Z 752.657,A -85,B 0,C 180,E1 8217.672,E2 8217.672} C_VEL
LIN {X 0,Y 163.699,Z 757.11,A -85,B 0,C 180,E1 8211.496,E2 8211.496} C_VEL
LIN {X 0,Y 161.245,Z 760.229,A -85,B 0,C 180,E1 8205.463,E2 8205.463} C_VEL
LIN {X 0,Y 160.133,Z 762.312,A -85,B 0,C 180,E1 8199.342,E2 8199.342} C_VEL
LIN {X 0,Y 159.963,Z 763.311,A -85,B 0,C 180,E1 8193.942,E2 8193.942} C_VEL
LIN {X 0,Y 159.996,Z 763.522,A -85,B 0,C 180,E1 8188.568,E2 8188.568} C_VEL
LIN {X 0,Y 160.014,Z 762.761,A -85,B 0,C 180,E1 8182.461,E2 8182.461} C_VEL
LIN {X 0,Y 160.922,Z 760.742,A -85,B 0,C 180,E1 8175.77,E2 8175.77} C_VEL
LIN {X 0,Y 163.162,Z 757.74,A -85,B 0,C 180,E1 8169.558,E2 8169.558} C_VEL
LIN {X 0,Y 166.834,Z 753.742,A -85,B 0,C 180,E1 8163.676,E2 8163.676} C_VEL
LIN {X 0,Y 171.986,Z 748.643,A -85,B 0,C 180,E1 8158.063,E2 8158.063} C_VEL
LIN {X 0,Y 178.573,Z 742.386,A -85,B 0,C 180,E1 8152.797,E2 8152.797} C_VEL
LIN {X 0,Y 186.487,Z 734.898,A -85,B 0,C 180,E1 8147.923,E2 8147.923} C_VEL
LIN {X 0,Y 197.324,Z 724.452,A -85,B 0,C 180,E1 8142.722,E2 8142.722} C_VEL
LIN {X 0,Y 208.934,Z 712.364,A -85,B 0,C 180,E1 8138.303,E2 8138.303} C_VEL
LIN {X 0,Y 219.09,Z 701.124,A -85,B 0,C 180,E1 8135.103,E2 8135.103} C_VEL
LIN {X 0,Y 228.738,Z 689.664,A -85,B 0,C 180,E1 8132.483,E2 8132.483} C_VEL
LIN {X 0,Y 238.673,Z 676.888,A -85,B 0,C 180,E1 8130.119,E2 8130.119} C_VEL
LIN {X 0,Y 248.601,Z 662.924,A -85,B 0,C 180,E1 8128.027,E2 8128.027} C_VEL
LIN {X 0,Y 260.463,Z 644.265,A -85,B 0,C 180,E1 8125.829,E2 8125.829} C_VEL
LIN {X 0,Y 269.798,Z 627.349,A -85,B 0,C 180,E1 8124.277,E2 8124.277} C_VEL
LIN {X 0,Y 277.669,Z 611.222,A -85,B 0,C 180,E1 8123.084,E2 8123.084} C_VEL
LIN {X 0,Y 284.391,Z 595.506,A -85,B 0,C 180,E1 8122.133,E2 8122.133} C_VEL
LIN {X 0,Y 290.35,Z 579.442,A -85,B 0,C 180,E1 8121.345,E2 8121.345} C_VEL
LIN {X 0,Y 295.505,Z 563.07,A -85,B 0,C 180,E1 8120.698,E2 8120.698} C_VEL
LIN {X 0,Y 300.098,Z 545.328,A -85,B 0,C 180,E1 8120.15,E2 8120.15} C_VEL
LIN {X 0,Y 304.473,Z 522.972,A -85,B 0,C 180,E1 8119.615,E2 8119.615} C_VEL
LIN {X 0,Y 308.295,Z 488.856,A -85,B 0,C 180,E1 8119.014,E2 8119.014} C_VEL
LIN {X 0,Y 316.421,Z 407.027,A -85,B 0,C 180,E1 8117.66,E2 8117.66} C_VEL
LIN {X 0,Y 312.833,Z 399.162,A -85,B 0,C 180,E1 8114.815,E2 8114.815} C_VEL
LIN {X 0,Y 309.324,Z 392.084,A -85,B 0,C 180,E1 8111.372,E2 8111.372} C_VEL
LIN {X 0,Y 307.304,Z 388.208,A -85,B 0,C 180,E1 8108.797,E2 8108.797} C_VEL
LIN {X 0,Y 305.653,Z 384.702,A -85,B 0,C 180,E1 8105.821,E2 8105.821} C_VEL
LIN {X 0,Y 304.326,Z 381.987,A -85,B 0,C 180,E1 8099.812,E2 8099.812} C_VEL
LIN {X 0,Y 305.862,Z 385.083,A -85,B 0,C 180,E1 8093.43,E2 8093.43} C_VEL
LIN {X 0,Y 308.16,Z 389.861,A -85,B 0,C 180,E1 8089.72,E2 8089.72} C_VEL
LIN {X 0,Y 310.48,Z 394.508,A -85,B 0,C 180,E1 8087.066,E2 8087.066} C_VEL
LIN {X 0,Y 313.538,Z 400.718,A -85,B 0,C 180,E1 8084.272,E2 8084.272} C_VEL
LIN {X 0,Y 317.572,Z 409.586,A -85,B 0,C 180,E1 8081.22,E2 8081.22} C_VEL
LIN {X 0,Y 321.879,Z 419.726,A -85,B 0,C 180,E1 8078.449,E2 8078.449} C_VEL
LIN {X 0,Y 330.853,Z 437.261,A -85,B 0,C 180,E1 8073.914,E2 8073.914} C_VEL
LIN {X 0,Y 344.243,Z 455.581,A -85,B 0,C 180,E1 8068.916,E2 8068.916} C_VEL
LIN {X 0,Y 365.545,Z 476.472,A -85,B 0,C 180,E1 8063.052,E2 8063.052} C_VEL
LIN {X 0,Y 390.021,Z 495.656,A -85,B 0,C 180,E1 8057.902,E2 8057.902} C_VEL
LIN {X 0,Y 401.499,Z 504.28,A -85,B 0,C 180,E1 8055.489,E2 8055.489} C_VEL
LIN {X 0,Y 411.358,Z 511.942,A -85,B 0,C 180,E1 8053.179,E2 8053.179} C_VEL
LIN {X 0,Y 420.156,Z 518.773,A -85,B 0,C 180,E1 8050.923,E2 8050.923} C_VEL
LIN {X 0,Y 429.799,Z 526.191,A -85,B 0,C 180,E1 8048.264,E2 8048.264} C_VEL
LIN {X 0,Y 438.223,Z 532.801,A -85,B 0,C 180,E1 8045.792,E2 8045.792} C_VEL
LIN {X 0,Y 446.918,Z 539.707,A -85,B 0,C 180,E1 8043.081,E2 8043.081} C_VEL
LIN {X 0,Y 454.655,Z 545.406,A -85,B 0,C 180,E1 8040.528,E2 8040.528} C_VEL
LIN {X 0,Y 461.272,Z 550.488,A -85,B 0,C 180,E1 8038.196,E2 8038.196} C_VEL
LIN {X 0,Y 467.616,Z 554.997,A -85,B 0,C 180,E1 8035.813,E2 8035.813} C_VEL
LIN {X 0,Y 473.554,Z 559.591,A -85,B 0,C 180,E1 8033.385,E2 8033.385} C_VEL
LIN {X 0,Y 479.734,Z 563.557,A -85,B 0,C 180,E1 8030.621,E2 8030.621} C_VEL
LIN {X 0,Y 484.489,Z 567.544,A -85,B 0,C 180,E1 8028.155,E2 8028.155} C_VEL
LIN {X 0,Y 488.841,Z 570.524,A -85,B 0,C 180,E1 8025.662,E2 8025.662} C_VEL
LIN {X 0,Y 492.9,Z 572.679,A -85,B 0,C 180,E1 8023.011,E2 8023.011} C_VEL
LIN {X 0,Y 494.78,Z 574.028,A -85,B 0,C 180,E1 8021.539,E2 8021.539} C_VEL
LIN {X 0,Y 497.348,Z 576.457,A -85,B 0,C 180,E1 8019.021,E2 8019.021} C_VEL
LIN {X 0,Y 499.402,Z 578.114,A -85,B 0,C 180,E1 8016.552,E2 8016.552} C_VEL
LIN {X 0,Y 500.763,Z 579.134,A -85,B 0,C 180,E1 8014.007,E2 8014.007} C_VEL
LIN {X 0,Y 501.533,Z 579.612,A -85,B 0,C 180,E1 8011.371,E2 8011.371} C_VEL
LIN {X 0,Y 501.554,Z 579.62,A -85,B 0,C 180,E1 8008.858,E2 8008.858} C_VEL
LIN {X 0,Y 500.817,Z 579.171,A -85,B 0,C 180,E1 8006.108,E2 8006.108} C_VEL
LIN {X 0,Y 499.472,Z 578.169,A -85,B 0,C 180,E1 8003.564,E2 8003.564} C_VEL
LIN {X 0,Y 497.474,Z 576.561,A -85,B 0,C 180,E1 8001.098,E2 8001.098} C_VEL
LIN {X 0,Y 494.845,Z 574.1,A -85,B 0,C 180,E1 7998.522,E2 7998.522} C_VEL
LIN {X 0,Y 493.067,Z 572.756,A -85,B 0,C 180,E1 7997.112,E2 7997.112} C_VEL
LIN {X 0,Y 489.256,Z 570.768,A -85,B 0,C 180,E1 7994.595,E2 7994.595} C_VEL
LIN {X 0,Y 485.008,Z 567.919,A -85,B 0,C 180,E1 7992.113,E2 7992.113} C_VEL
LIN {X 0,Y 480.131,Z 563.919,A -85,B 0,C 180,E1 7989.577,E2 7989.577} C_VEL
LIN {X 0,Y 474.106,Z 559.977,A -85,B 0,C 180,E1 7986.857,E2 7986.857} C_VEL
LIN {X 0,Y 468.466,Z 555.727,A -85,B 0,C 180,E1 7984.536,E2 7984.536} C_VEL
LIN {X 0,Y 463.89,Z 552.258,A -85,B 0,C 180,E1 7982.764,E2 7982.764} C_VEL
LIN {X 0,Y 456.771,Z 547.132,A -85,B 0,C 180,E1 7980.209,E2 7980.209} C_VEL
LIN {X 0,Y 450.614,Z 542.4,A -85,B 0,C 180,E1 7978.127,E2 7978.127} C_VEL
LIN {X 0,Y 442.581,Z 536.265,A -85,B 0,C 180,E1 7975.55,E2 7975.55} C_VEL
LIN {X 0,Y 433.796,Z 529.454,A -85,B 0,C 180,E1 7972.895,E2 7972.895} C_VEL
LIN {X 0,Y 425.004,Z 522.568,A -85,B 0,C 180,E1 7970.396,E2 7970.396} C_VEL
LIN {X 0,Y 415.699,Z 515.159,A -85,B 0,C 180,E1 7967.906,E2 7967.906} C_VEL
LIN {X 0,Y 406.517,Z 508.12,A -85,B 0,C 180,E1 7965.655,E2 7965.655} C_VEL
LIN {X 0,Y 396.847,Z 500.828,A -85,B 0,C 180,E1 7963.51,E2 7963.51} C_VEL
LIN {X 0,Y 388.064,Z 494.258,A -85,B 0,C 180,E1 7961.714,E2 7961.714} C_VEL
LIN {X 0,Y 360.798,Z 472.209,A -85,B 0,C 180,E1 7955.786,E2 7955.786} C_VEL
LIN {X 0,Y 342.772,Z 453.81,A -85,B 0,C 180,E1 7950.599,E2 7950.599} C_VEL
LIN {X 0,Y 329.843,Z 435.603,A -85,B 0,C 180,E1 7945.641,E2 7945.641} C_VEL
LIN {X 0,Y 320.747,Z 417.061,A -85,B 0,C 180,E1 7940.865,E2 7940.865} C_VEL
LIN {X 0,Y 316.821,Z 407.918,A -85,B 0,C 180,E1 7938.254,E2 7938.254} C_VEL
LIN {X 0,Y 312.808,Z 399.101,A -85,B 0,C 180,E1 7935.101,E2 7935.101} C_VEL
LIN {X 0,Y 309.386,Z 392.187,A -85,B 0,C 180,E1 7931.748,E2 7931.748} C_VEL
LIN {X 0,Y 307.352,Z 388.291,A -85,B 0,C 180,E1 7929.173,E2 7929.173} C_VEL
LIN {X 0,Y 305.687,Z 384.737,A -85,B 0,C 180,E1 7926.197,E2 7926.197} C_VEL
LIN {X 0,Y 304.326,Z 381.987,A -85,B 0,C 180,E1 7920.188,E2 7920.188} C_VEL
LIN {X 0,Y 305.836,Z 384.96,A -85,B 0,C 180,E1 7913.806,E2 7913.806} C_VEL
LIN {X 0,Y 308.108,Z 389.749,A -85,B 0,C 180,E1 7910.096,E2 7910.096} C_VEL
LIN {X 0,Y 310.325,Z 394.199,A -85,B 0,C 180,E1 7907.533,E2 7907.533} C_VEL
LIN {X 0,Y 313.565,Z 400.765,A -85,B 0,C 180,E1 7904.558,E2 7904.558} C_VEL
LIN {X 0,Y 316.441,Z 407.168,A -85,B 0,C 180,E1 7902.319,E2 7902.319} C_VEL
LIN {X 0,Y 305.288,Z 516.721,A -85,B 0,C 180,E1 7900.504,E2 7900.504} C_VEL
LIN {X 0,Y 301.446,Z 539.643,A -85,B 0,C 180,E1 7900.004,E2 7900.004} C_VEL
LIN {X 0,Y 296.157,Z 560.843,A -85,B 0,C 180,E1 7899.378,E2 7899.378} C_VEL
LIN {X 0,Y 290.777,Z 578.199,A -85,B 0,C 180,E1 7898.71,E2 7898.71} C_VEL
LIN {X 0,Y 284.813,Z 594.445,A -85,B 0,C 180,E1 7897.925,E2 7897.925} C_VEL
LIN {X 0,Y 278.086,Z 610.302,A -85,B 0,C 180,E1 7896.977,E2 7896.977} C_VEL
LIN {X 0,Y 270.621,Z 625.739,A -85,B 0,C 180,E1 7895.852,E2 7895.852} C_VEL
LIN {X 0,Y 262.472,Z 640.713,A -85,B 0,C 180,E1 7894.519,E2 7894.519} C_VEL
LIN {X 0,Y 252.909,Z 656.437,A -85,B 0,C 180,E1 7892.801,E2 7892.801} C_VEL
LIN {X 0,Y 240.151,Z 674.93,A -85,B 0,C 180,E1 7890.207,E2 7890.207} C_VEL
LIN {X 0,Y 230.187,Z 687.886,A -85,B 0,C 180,E1 7887.879,E2 7887.879} C_VEL
LIN {X 0,Y 220.271,Z 699.768,A -85,B 0,C 180,E1 7885.236,E2 7885.236} C_VEL
LIN {X 0,Y 210.382,Z 710.79,A -85,B 0,C 180,E1 7882.186,E2 7882.186} C_VEL
LIN {X 0,Y 200.854,Z 720.768,A -85,B 0,C 180,E1 7878.729,E2 7878.729} C_VEL
LIN {X 0,Y 191.17,Z 730.414,A -85,B 0,C 180,E1 7874.489,E2 7874.489} C_VEL
LIN {X 0,Y 179.878,Z 741.185,A -85,B 0,C 180,E1 7868.092,E2 7868.092} C_VEL
LIN {X 0,Y 174.322,Z 746.487,A -85,B 0,C 180,E1 7863.976,E2 7863.976} C_VEL
LIN {X 0,Y 170.805,Z 748.934,A -85,B 0,C 180,E1 7861.82,E2 7861.82} C_VEL
LIN {X 0,Y 161.567,Z 753.535,A -85,B 0,C 180,E1 7857.495,E2 7857.495} C_VEL
LIN {X 0,Y 157.602,Z 755.686,A -85,B 0,C 180,E1 7854.734,E2 7854.734} C_VEL
LIN {X 0,Y 156.851,Z 756.246,A -85,B 0,C 180,E1 7853.783,E2 7853.783} C_VEL
LIN {X 0,Y 153.553,Z 759.902,A -85,B 0,C 180,E1 7846.647,E2 7846.647} C_VEL
LIN {X 0,Y 152.214,Z 762.046,A -85,B 0,C 180,E1 7840.215,E2 7840.215} C_VEL
LIN {X 0,Y 151.962,Z 763.136,A -85,B 0,C 180,E1 7834.15,E2 7834.15} C_VEL
LIN {X 0,Y 152.002,Z 763.377,A -85,B 0,C 180,E1 7828.869,E2 7828.869} C_VEL
LIN {X 0,Y 152.033,Z 762.585,A -85,B 0,C 180,E1 7822.062,E2 7822.062} C_VEL
LIN {X 0,Y 153.02,Z 760.65,A -85,B 0,C 180,E1 7815.238,E2 7815.238} C_VEL
LIN {X 0,Y 155.558,Z 757.562,A -85,B 0,C 180,E1 7808.51,E2 7808.51} C_VEL
LIN {X 0,Y 159.558,Z 753.563,A -85,B 0,C 180,E1 7802.376,E2 7802.376} C_VEL
LIN {X 0,Y 165.106,Z 748.464,A -85,B 0,C 180,E1 7796.563,E2 7796.563} C_VEL
LIN {X 0,Y 171.677,Z 742.608,A -85,B 0,C 180,E1 7791.456,E2 7791.456} C_VEL
LIN {X 0,Y 179.449,Z 735.657,A -85,B 0,C 180,E1 7786.744,E2 7786.744} C_VEL
LIN {X 0,Y 188.299,Z 727.526,A -85,B 0,C 180,E1 7782.438,E2 7782.438} C_VEL
LIN {X 0,Y 198.738,Z 717.495,A -85,B 0,C 180,E1 7778.302,E2 7778.302} C_VEL
LIN {X 0,Y 212.191,Z 703.546,A -85,B 0,C 180,E1 7773.98,E2 7773.98} C_VEL
LIN {X 0,Y 223.565,Z 690.577,A -85,B 0,C 180,E1 7770.953,E2 7770.953} C_VEL
LIN {X 0,Y 233.548,Z 678.208,A -85,B 0,C 180,E1 7768.652,E2 7768.652} C_VEL
LIN {X 0,Y 242.909,Z 665.548,A -85,B 0,C 180,E1 7766.732,E2 7766.732} C_VEL
LIN {X 0,Y 252.138,Z 651.851,A -85,B 0,C 180,E1 7765.038,E2 7765.038} C_VEL
LIN {X 0,Y 261.163,Z 636.983,A -85,B 0,C 180,E1 7763.534,E2 7763.534} C_VEL
LIN {X 0,Y 271.223,Z 618.313,A -85,B 0,C 180,E1 7762.02,E2 7762.02} C_VEL
LIN {X 0,Y 280.171,Z 598.515,A -85,B 0,C 180,E1 7760.786,E2 7760.786} C_VEL
LIN {X 0,Y 286.653,Z 581.753,A -85,B 0,C 180,E1 7759.961,E2 7759.961} C_VEL
LIN {X 0,Y 292.105,Z 565.123,A -85,B 0,C 180,E1 7759.304,E2 7759.304} C_VEL
LIN {X 0,Y 296.803,Z 547.75,A -85,B 0,C 180,E1 7758.769,E2 7758.769} C_VEL
LIN {X 0,Y 300.497,Z 530.331,A -85,B 0,C 180,E1 7758.347,E2 7758.347} C_VEL
LIN {X 0,Y 303.261,Z 512.065,A -85,B 0,C 180,E1 7757.984,E2 7757.984} C_VEL
LIN {X 0,Y 313.572,Z 411.879,A -85,B 0,C 180,E1 7756.348,E2 7756.348} C_VEL
LIN {X 0,Y 310.268,Z 404.637,A -85,B 0,C 180,E1 7753.464,E2 7753.464} C_VEL
LIN {X 0,Y 307.537,Z 398.934,A -85,B 0,C 180,E1 7750.491,E2 7750.491} C_VEL
LIN {X 0,Y 306.064,Z 395.907,A -85,B 0,C 180,E1 7748.454,E2 7748.454} C_VEL
LIN {X 0,Y 304.498,Z 392.497,A -85,B 0,C 180,E1 7745.465,E2 7745.465} C_VEL
LIN {X 0,Y 303.351,Z 389.928,A -85,B 0,C 180,E1 7739.811,E2 7739.811} C_VEL
LIN {X 0,Y 304.782,Z 393.033,A -85,B 0,C 180,E1 7733.596,E2 7733.596} C_VEL
LIN {X 0,Y 306.883,Z 397.56,A -85,B 0,C 180,E1 7730.056,E2 7730.056} C_VEL
LIN {X 0,Y 309.119,Z 402.229,A -85,B 0,C 180,E1 7727.389,E2 7727.389} C_VEL
LIN {X 0,Y 312.293,Z 408.984,A -85,B 0,C 180,E1 7724.398,E2 7724.398} C_VEL
LIN {X 0,Y 316.626,Z 419.104,A -85,B 0,C 180,E1 7721.066,E2 7721.066} C_VEL
LIN {X 0,Y 327.465,Z 442.636,A -85,B 0,C 180,E1 7714.886,E2 7714.886} C_VEL
LIN {X 0,Y 340.252,Z 460.964,A -85,B 0,C 180,E1 7709.833,E2 7709.833} C_VEL
LIN {X 0,Y 356.744,Z 478.091,A -85,B 0,C 180,E1 7704.93,E2 7704.93} C_VEL
LIN {X 0,Y 384.111,Z 500.64,A -85,B 0,C 180,E1 7698.807,E2 7698.807} C_VEL
LIN {X 0,Y 394.937,Z 508.716,A -85,B 0,C 180,E1 7696.595,E2 7696.595} C_VEL
LIN {X 0,Y 404.732,Z 516.169,A -85,B 0,C 180,E1 7694.385,E2 7694.385} C_VEL
LIN {X 0,Y 414.306,Z 523.404,A -85,B 0,C 180,E1 7692.036,E2 7692.036} C_VEL
LIN {X 0,Y 423.444,Z 530.628,A -85,B 0,C 180,E1 7689.603,E2 7689.603} C_VEL
LIN {X 0,Y 432.611,Z 537.787,A -85,B 0,C 180,E1 7687.008,E2 7687.008} C_VEL
LIN {X 0,Y 440.536,Z 543.869,A -85,B 0,C 180,E1 7684.637,E2 7684.637} C_VEL
LIN {X 0,Y 448.086,Z 549.616,A -85,B 0,C 180,E1 7682.25,E2 7682.25} C_VEL
LIN {X 0,Y 454.728,Z 554.621,A -85,B 0,C 180,E1 7680.044,E2 7680.044} C_VEL
LIN {X 0,Y 461.762,Z 559.728,A -85,B 0,C 180,E1 7677.522,E2 7677.522} C_VEL
LIN {X 0,Y 466.064,Z 562.872,A -85,B 0,C 180,E1 7675.889,E2 7675.889} C_VEL
LIN {X 0,Y 471.879,Z 567.319,A -85,B 0,C 180,E1 7673.532,E2 7673.532} C_VEL
LIN {X 0,Y 477.744,Z 570.947,A -85,B 0,C 180,E1 7670.968,E2 7670.968} C_VEL
LIN {X 0,Y 482.894,Z 575.247,A -85,B 0,C 180,E1 7668.342,E2 7668.342} C_VEL
LIN {X 0,Y 487.365,Z 578.317,A -85,B 0,C 180,E1 7665.8,E2 7665.8} C_VEL
LIN {X 0,Y 491.427,Z 580.487,A -85,B 0,C 180,E1 7663.171,E2 7663.171} C_VEL
LIN {X 0,Y 493.355,Z 581.801,A -85,B 0,C 180,E1 7661.692,E2 7661.692} C_VEL
LIN {X 0,Y 496.122,Z 584.374,A -85,B 0,C 180,E1 7659.043,E2 7659.043} C_VEL
LIN {X 0,Y 498.221,Z 586.073,A -85,B 0,C 180,E1 7656.452,E2 7656.452} C_VEL
LIN {X 0,Y 499.615,Z 587.105,A -85,B 0,C 180,E1 7653.786,E2 7653.786} C_VEL
LIN {X 0,Y 500.308,Z 587.518,A -85,B 0,C 180,E1 7651.26,E2 7651.26} C_VEL
LIN {X 0,Y 500.331,Z 587.524,A -85,B 0,C 180,E1 7648.741,E2 7648.741} C_VEL
LIN {X 0,Y 499.557,Z 587.044,A -85,B 0,C 180,E1 7645.983,E2 7645.983} C_VEL
LIN {X 0,Y 498.029,Z 585.951,A -85,B 0,C 180,E1 7643.314,E2 7643.314} C_VEL
LIN {X 0,Y 496.017,Z 584.268,A -85,B 0,C 180,E1 7640.838,E2 7640.838} C_VEL
LIN {X 0,Y 493.193,Z 581.651,A -85,B 0,C 180,E1 7638.186,E2 7638.186} C_VEL
LIN {X 0,Y 491.053,Z 580.315,A -85,B 0,C 180,E1 7636.579,E2 7636.579} C_VEL
LIN {X 0,Y 486.88,Z 578.018,A -85,B 0,C 180,E1 7633.906,E2 7633.906} C_VEL
LIN {X 0,Y 482.288,Z 574.792,A -85,B 0,C 180,E1 7631.346,E2 7631.346} C_VEL
LIN {X 0,Y 477.1,Z 570.592,A -85,B 0,C 180,E1 7628.745,E2 7628.745} C_VEL
LIN {X 0,Y 471.157,Z 566.807,A -85,B 0,C 180,E1 7626.159,E2 7626.159} C_VEL
LIN {X 0,Y 464.432,Z 561.448,A -85,B 0,C 180,E1 7623.45,E2 7623.45} C_VEL
LIN {X 0,Y 457.497,Z 556.779,A -85,B 0,C 180,E1 7620.954,E2 7620.954} C_VEL
LIN {X 0,Y 450.09,Z 550.953,A -85,B 0,C 180,E1 7618.385,E2 7618.385} C_VEL
LIN {X 0,Y 442.235,Z 545.257,A -85,B 0,C 180,E1 7615.899,E2 7615.899} C_VEL
LIN {X 0,Y 434.262,Z 539.034,A -85,B 0,C 180,E1 7613.473,E2 7613.473} C_VEL
LIN {X 0,Y 424.769,Z 531.582,A -85,B 0,C 180,E1 7610.756,E2 7610.756} C_VEL
LIN {X 0,Y 415.683,Z 524.559,A -85,B 0,C 180,E1 7608.321,E2 7608.321} C_VEL
LIN {X 0,Y 405.655,Z 516.898,A -85,B 0,C 180,E1 7605.83,E2 7605.83} C_VEL
LIN {X 0,Y 396.113,Z 509.606,A -85,B 0,C 180,E1 7603.661,E2 7603.661} C_VEL
LIN {X 0,Y 386.057,Z 502.068,A -85,B 0,C 180,E1 7601.582,E2 7601.582} C_VEL
LIN {X 0,Y 358.319,Z 479.602,A -85,B 0,C 180,E1 7595.481,E2 7595.481} C_VEL
LIN {X 0,Y 340.142,Z 460.828,A -85,B 0,C 180,E1 7590.129,E2 7590.129} C_VEL
LIN {X 0,Y 327.377,Z 442.484,A -85,B 0,C 180,E1 7585.073,E2 7585.073} C_VEL
LIN {X 0,Y 318.493,Z 423.798,A -85,B 0,C 180,E1 7580.203,E2 7580.203} C_VEL
LIN {X 0,Y 314.795,Z 414.804,A -85,B 0,C 180,E1 7577.611,E2 7577.611} C_VEL
LIN {X 0,Y 311.173,Z 406.469,A -85,B 0,C 180,E1 7574.61,E2 7574.61} C_VEL
LIN {X 0,Y 307.904,Z 399.603,A -85,B 0,C 180,E1 7571.236,E2 7571.236} C_VEL
LIN {X 0,Y 306.11,Z 395.992,A -85,B 0,C 180,E1 7568.831,E2 7568.831} C_VEL
LIN {X 0,Y 304.531,Z 392.533,A -85,B 0,C 180,E1 7565.842,E2 7565.842} C_VEL
LIN {X 0,Y 303.351,Z 389.941,A -85,B 0,C 180,E1 7560,E2 7560} C_VEL
LIN {X 0,Y 304.794,Z 393.042,A -85,B 0,C 180,E1 7553.88,E2 7553.88} C_VEL
LIN {X 0,Y 306.833,Z 397.447,A -85,B 0,C 180,E1 7550.433,E2 7550.433} C_VEL
LIN {X 0,Y 308.967,Z 401.922,A -85,B 0,C 180,E1 7547.857,E2 7547.857} C_VEL
LIN {X 0,Y 312.266,Z 408.919,A -85,B 0,C 180,E1 7544.73,E2 7544.73} C_VEL
LIN {X 0,Y 313.565,Z 412.206,A -85,B 0,C 180,E1 7543.63,E2 7543.63} C_VEL
LIN {X 0,Y 302.677,Z 516.771,A -85,B 0,C 180,E1 7541.931,E2 7541.931} C_VEL
LIN {X 0,Y 298.716,Z 539.842,A -85,B 0,C 180,E1 7541.439,E2 7541.439} C_VEL
LIN {X 0,Y 293.206,Z 561.41,A -85,B 0,C 180,E1 7540.82,E2 7540.82} C_VEL
LIN {X 0,Y 287.957,Z 578.023,A -85,B 0,C 180,E1 7540.2,E2 7540.2} C_VEL
LIN {X 0,Y 281.888,Z 594.269,A -85,B 0,C 180,E1 7539.441,E2 7539.441} C_VEL
LIN {X 0,Y 275.035,Z 610.126,A -85,B 0,C 180,E1 7538.522,E2 7538.522} C_VEL
LIN {X 0,Y 267.422,Z 625.562,A -85,B 0,C 180,E1 7537.429,E2 7537.429} C_VEL
LIN {X 0,Y 259.097,Z 640.536,A -85,B 0,C 180,E1 7536.133,E2 7536.133} C_VEL
LIN {X 0,Y 249.311,Z 656.26,A -85,B 0,C 180,E1 7534.457,E2 7534.457} C_VEL
LIN {X 0,Y 236.253,Z 674.714,A -85,B 0,C 180,E1 7531.922,E2 7531.922} C_VEL
LIN {X 0,Y 225.969,Z 687.708,A -85,B 0,C 180,E1 7529.625,E2 7529.625} C_VEL
LIN {X 0,Y 215.731,Z 699.591,A -85,B 0,C 180,E1 7527.014,E2 7527.014} C_VEL
LIN {X 0,Y 205.993,Z 710.082,A -85,B 0,C 180,E1 7524.145,E2 7524.145} C_VEL
LIN {X 0,Y 196.191,Z 719.97,A -85,B 0,C 180,E1 7520.765,E2 7520.765} C_VEL
LIN {X 0,Y 186.563,Z 729.152,A -85,B 0,C 180,E1 7516.785,E2 7516.785} C_VEL
LIN {X 0,Y 176.405,Z 738.471,A -85,B 0,C 180,E1 7511.535,E2 7511.535} C_VEL
LIN {X 0,Y 166.501,Z 747.237,A -85,B 0,C 180,E1 7504.64,E2 7504.64} C_VEL
LIN {X 0,Y 160.425,Z 752.75,A -85,B 0,C 180,E1 7498.676,E2 7498.676} C_VEL
LIN {X 0,Y 156.851,Z 756.246,A -85,B 0,C 180,E1 7493.783,E2 7493.783} C_VEL
LIN {X 0,Y 154.373,Z 757.83,A -85,B 0,C 180,E1 7491.132,E2 7491.132} C_VEL
LIN {X 0,Y 148.431,Z 760.048,A -85,B 0,C 180,E1 7486.649,E2 7486.649} C_VEL
LIN {X 0,Y 144.84,Z 761.43,A -85,B 0,C 180,E1 7482.774,E2 7482.774} C_VEL
LIN {X 0,Y 144.327,Z 761.764,A -85,B 0,C 180,E1 7481.248,E2 7481.248} C_VEL
LIN {X 0,Y 143.958,Z 762.93,A -85,B 0,C 180,E1 7474.78,E2 7474.78} C_VEL
LIN {X 0,Y 144.002,Z 763.202,A -85,B 0,C 180,E1 7468.807,E2 7468.807} C_VEL
LIN {X 0,Y 144.06,Z 762.409,A -85,B 0,C 180,E1 7461.62,E2 7461.62} C_VEL
LIN {X 0,Y 145.192,Z 760.473,A -85,B 0,C 180,E1 7454.422,E2 7454.422} C_VEL
LIN {X 0,Y 148.01,Z 757.384,A -85,B 0,C 180,E1 7447.355,E2 7447.355} C_VEL
LIN {X 0,Y 152.372,Z 753.385,A -85,B 0,C 180,E1 7440.953,E2 7440.953} C_VEL
LIN {X 0,Y 158.346,Z 748.285,A -85,B 0,C 180,E1 7434.932,E2 7434.932} C_VEL
LIN {X 0,Y 165.839,Z 742.029,A -85,B 0,C 180,E1 7429.377,E2 7429.377} C_VEL
LIN {X 0,Y 174.691,Z 734.54,A -85,B 0,C 180,E1 7424.326,E2 7424.326} C_VEL
LIN {X 0,Y 186.621,Z 724.095,A -85,B 0,C 180,E1 7419.033,E2 7419.033} C_VEL
LIN {X 0,Y 199.234,Z 712.007,A -85,B 0,C 180,E1 7414.619,E2 7414.619} C_VEL
LIN {X 0,Y 209.936,Z 700.995,A -85,B 0,C 180,E1 7411.523,E2 7411.523} C_VEL
LIN {X 0,Y 219.666,Z 690.198,A -85,B 0,C 180,E1 7409.092,E2 7409.092} C_VEL
LIN {X 0,Y 229.764,Z 678.031,A -85,B 0,C 180,E1 7406.875,E2 7406.875} C_VEL
LIN {X 0,Y 239.372,Z 665.371,A -85,B 0,C 180,E1 7404.999,E2 7404.999} C_VEL
LIN {X 0,Y 248.82,Z 651.674,A -85,B 0,C 180,E1 7403.349,E2 7403.349} C_VEL
LIN {X 0,Y 258.043,Z 636.807,A -85,B 0,C 180,E1 7401.888,E2 7401.888} C_VEL
LIN {X 0,Y 268.304,Z 618.137,A -85,B 0,C 180,E1 7400.424,E2 7400.424} C_VEL
LIN {X 0,Y 277.416,Z 598.339,A -85,B 0,C 180,E1 7399.231,E2 7399.231} C_VEL
LIN {X 0,Y 284.01,Z 581.577,A -85,B 0,C 180,E1 7398.436,E2 7398.436} C_VEL
LIN {X 0,Y 289.551,Z 564.948,A -85,B 0,C 180,E1 7397.805,E2 7397.805} C_VEL
LIN {X 0,Y 294.348,Z 547.465,A -85,B 0,C 180,E1 7397.288,E2 7397.288} C_VEL
LIN {X 0,Y 298.115,Z 529.916,A -85,B 0,C 180,E1 7396.879,E2 7396.879} C_VEL
LIN {X 0,Y 300.949,Z 511.376,A -85,B 0,C 180,E1 7396.523,E2 7396.523} C_VEL
LIN {X 0,Y 310.86,Z 416.89,A -85,B 0,C 180,E1 7395.007,E2 7395.007} C_VEL
LIN {X 0,Y 307.872,Z 410.163,A -85,B 0,C 180,E1 7392.092,E2 7392.092} C_VEL
LIN {X 0,Y 305.762,Z 405.598,A -85,B 0,C 180,E1 7389.506,E2 7389.506} C_VEL
LIN {X 0,Y 304.661,Z 403.297,A -85,B 0,C 180,E1 7387.828,E2 7387.828} C_VEL
LIN {X 0,Y 303.438,Z 400.379,A -85,B 0,C 180,E1 7385.294,E2 7385.294} C_VEL
LIN {X 0,Y 302.376,Z 397.87,A -85,B 0,C 180,E1 7379.811,E2 7379.811} C_VEL
LIN {X 0,Y 303.664,Z 400.839,A -85,B 0,C 180,E1 7373.866,E2 7373.866} C_VEL
LIN {X 0,Y 305.617,Z 405.258,A -85,B 0,C 180,E1 7370.395,E2 7370.395} C_VEL
LIN {X 0,Y 307.852,Z 410.121,A -85,B 0,C 180,E1 7367.622,E2 7367.622} C_VEL
LIN {X 0,Y 310.785,Z 416.725,A -85,B 0,C 180,E1 7364.751,E2 7364.751} C_VEL
LIN {X 0,Y 314.801,Z 426.59,A -85,B 0,C 180,E1 7361.529,E2 7361.529} C_VEL
LIN {X 0,Y 324.515,Z 448.6,A -85,B 0,C 180,E1 7355.711,E2 7355.711} C_VEL
LIN {X 0,Y 336.46,Z 466.452,A -85,B 0,C 180,E1 7350.734,E2 7350.734} C_VEL
LIN {X 0,Y 352.224,Z 483.612,A -85,B 0,C 180,E1 7345.8,E2 7345.8} C_VEL
LIN {X 0,Y 379.822,Z 506.859,A -85,B 0,C 180,E1 7339.341,E2 7339.341} C_VEL
LIN {X 0,Y 390.794,Z 515.027,A -85,B 0,C 180,E1 7337.11,E2 7337.11} C_VEL
LIN {X 0,Y 401.588,Z 523.213,A -85,B 0,C 180,E1 7334.696,E2 7334.696} C_VEL
LIN {X 0,Y 411.004,Z 530.309,A -85,B 0,C 180,E1 7332.408,E2 7332.408} C_VEL
LIN {X 0,Y 420.443,Z 537.732,A -85,B 0,C 180,E1 7329.928,E2 7329.928} C_VEL
LIN {X 0,Y 430.11,Z 545.203,A -85,B 0,C 180,E1 7327.229,E2 7327.229} C_VEL
LIN {X 0,Y 438.072,Z 551.287,A -85,B 0,C 180,E1 7324.86,E2 7324.86} C_VEL
LIN {X 0,Y 446.403,Z 557.546,A -85,B 0,C 180,E1 7322.256,E2 7322.256} C_VEL
LIN {X 0,Y 453.813,Z 563.202,A -85,B 0,C 180,E1 7319.76,E2 7319.76} C_VEL
LIN {X 0,Y 461.269,Z 568.326,A -85,B 0,C 180,E1 7317.133,E2 7317.133} C_VEL
LIN {X 0,Y 468.434,Z 573.935,A -85,B 0,C 180,E1 7314.293,E2 7314.293} C_VEL
LIN {X 0,Y 474.679,Z 577.994,A -85,B 0,C 180,E1 7311.628,E2 7311.628} C_VEL
LIN {X 0,Y 479.243,Z 581.524,A -85,B 0,C 180,E1 7309.429,E2 7309.429} C_VEL
LIN {X 0,Y 484.076,Z 585.107,A -85,B 0,C 180,E1 7306.806,E2 7306.806} C_VEL
LIN {X 0,Y 488.338,Z 587.577,A -85,B 0,C 180,E1 7304.221,E2 7304.221} C_VEL
LIN {X 0,Y 491.478,Z 589.357,A -85,B 0,C 180,E1 7301.975,E2 7301.975} C_VEL
LIN {X 0,Y 494.316,Z 592.009,A -85,B 0,C 180,E1 7299.311,E2 7299.311} C_VEL
LIN {X 0,Y 496.482,Z 593.799,A -85,B 0,C 180,E1 7296.707,E2 7296.707} C_VEL
LIN {X 0,Y 497.925,Z 594.849,A -85,B 0,C 180,E1 7294.145,E2 7294.145} C_VEL
LIN {X 0,Y 498.736,Z 595.35,A -85,B 0,C 180,E1 7291.608,E2 7291.608} C_VEL
LIN {X 0,Y 498.807,Z 595.378,A -85,B 0,C 180,E1 7288.966,E2 7288.966} C_VEL
LIN {X 0,Y 498.157,Z 595.012,A -85,B 0,C 180,E1 7286.433,E2 7286.433} C_VEL
LIN {X 0,Y 496.806,Z 594.028,A -85,B 0,C 180,E1 7283.762,E2 7283.762} C_VEL
LIN {X 0,Y 494.644,Z 592.319,A -85,B 0,C 180,E1 7281.047,E2 7281.047} C_VEL
LIN {X 0,Y 492.043,Z 589.936,A -85,B 0,C 180,E1 7278.514,E2 7278.514} C_VEL
LIN {X 0,Y 490.152,Z 588.47,A -85,B 0,C 180,E1 7277.034,E2 7277.034} C_VEL
LIN {X 0,Y 486.311,Z 586.475,A -85,B 0,C 180,E1 7274.499,E2 7274.499} C_VEL
LIN {X 0,Y 481.767,Z 583.489,A -85,B 0,C 180,E1 7271.909,E2 7271.909} C_VEL
LIN {X 0,Y 476.844,Z 579.508,A -85,B 0,C 180,E1 7269.376,E2 7269.376} C_VEL
LIN {X 0,Y 470.561,Z 575.422,A -85,B 0,C 180,E1 7266.591,E2 7266.591} C_VEL
LIN {X 0,Y 464.347,Z 570.774,A -85,B 0,C 180,E1 7264.083,E2 7264.083} C_VEL
LIN {X 0,Y 460.079,Z 567.609,A -85,B 0,C 180,E1 7262.463,E2 7262.463} C_VEL
LIN {X 0,Y 453.795,Z 563.203,A -85,B 0,C 180,E1 7260.243,E2 7260.243} C_VEL
LIN {X 0,Y 446.393,Z 557.533,A -85,B 0,C 180,E1 7257.734,E2 7257.734} C_VEL
LIN {X 0,Y 438.491,Z 551.645,A -85,B 0,C 180,E1 7255.279,E2 7255.279} C_VEL
LIN {X 0,Y 432.021,Z 546.663,A -85,B 0,C 180,E1 7253.341,E2 7253.341} C_VEL
LIN {X 0,Y 422.165,Z 538.987,A -85,B 0,C 180,E1 7250.545,E2 7250.545} C_VEL
LIN {X 0,Y 413.005,Z 531.951,A -85,B 0,C 180,E1 7248.113,E2 7248.113} C_VEL
LIN {X 0,Y 403.052,Z 524.376,A -85,B 0,C 180,E1 7245.651,E2 7245.651} C_VEL
LIN {X 0,Y 393.632,Z 517.175,A -85,B 0,C 180,E1 7243.503,E2 7243.503} C_VEL
LIN {X 0,Y 383.008,Z 509.202,A -85,B 0,C 180,E1 7241.287,E2 7241.287} C_VEL
LIN {X 0,Y 356.243,Z 487.372,A -85,B 0,C 180,E1 7235.274,E2 7235.274} C_VEL
LIN {X 0,Y 337.535,Z 467.845,A -85,B 0,C 180,E1 7229.651,E2 7229.651} C_VEL
LIN {X 0,Y 325.029,Z 449.518,A -85,B 0,C 180,E1 7224.538,E2 7224.538} C_VEL
LIN {X 0,Y 316.408,Z 430.872,A -85,B 0,C 180,E1 7219.619,E2 7219.619} C_VEL
LIN {X 0,Y 312.981,Z 422.08,A -85,B 0,C 180,E1 7217.092,E2 7217.092} C_VEL
LIN {X 0,Y 309.464,Z 413.633,A -85,B 0,C 180,E1 7214.024,E2 7214.024} C_VEL
LIN {X 0,Y 306.448,Z 407.014,A -85,B 0,C 180,E1 7210.718,E2 7210.718} C_VEL
LIN {X 0,Y 304.82,Z 403.593,A -85,B 0,C 180,E1 7208.394,E2 7208.394} C_VEL
LIN {X 0,Y 303.47,Z 400.417,A -85,B 0,C 180,E1 7205.673,E2 7205.673} C_VEL
LIN {X 0,Y 302.375,Z 397.886,A -85,B 0,C 180,E1 7200,E2 7200} C_VEL
LIN {X 0,Y 303.679,Z 400.859,A -85,B 0,C 180,E1 7194.141,E2 7194.141} C_VEL
LIN {X 0,Y 305.569,Z 405.145,A -85,B 0,C 180,E1 7190.773,E2 7190.773} C_VEL
LIN {X 0,Y 307.703,Z 409.817,A -85,B 0,C 180,E1 7188.092,E2 7188.092} C_VEL
LIN {X 0,Y 310.759,Z 416.634,A -85,B 0,C 180,E1 7185.084,E2 7185.084} C_VEL
LIN {X 0,Y 310.851,Z 417.286,A -85,B 0,C 180,E1 7184.965,E2 7184.965} C_VEL
LIN {X 0,Y 300.285,Z 516.616,A -85,B 0,C 180,E1 7183.386,E2 7183.386} C_VEL
LIN {X 0,Y 296.236,Z 539.777,A -85,B 0,C 180,E1 7182.907,E2 7182.907} C_VEL
LIN {X 0,Y 290.669,Z 561.235,A -85,B 0,C 180,E1 7182.314,E2 7182.314} C_VEL
LIN {X 0,Y 285.335,Z 577.848,A -85,B 0,C 180,E1 7181.718,E2 7181.718} C_VEL
LIN {X 0,Y 278.982,Z 594.535,A -85,B 0,C 180,E1 7180.965,E2 7180.965} C_VEL
LIN {X 0,Y 272.189,Z 609.95,A -85,B 0,C 180,E1 7180.1,E2 7180.1} C_VEL
LIN {X 0,Y 264.431,Z 625.386,A -85,B 0,C 180,E1 7179.043,E2 7179.043} C_VEL
LIN {X 0,Y 255.933,Z 640.36,A -85,B 0,C 180,E1 7177.788,E2 7177.788} C_VEL
LIN {X 0,Y 245.928,Z 656.083,A -85,B 0,C 180,E1 7176.16,E2 7176.16} C_VEL
LIN {X 0,Y 232.87,Z 674.127,A -85,B 0,C 180,E1 7173.752,E2 7173.752} C_VEL
LIN {X 0,Y 221.968,Z 687.53,A -85,B 0,C 180,E1 7171.437,E2 7171.437} C_VEL
LIN {X 0,Y 211.407,Z 699.413,A -85,B 0,C 180,E1 7168.866,E2 7168.866} C_VEL
LIN {X 0,Y 201.324,Z 709.903,A -85,B 0,C 180,E1 7166.027,E2 7166.027} C_VEL
LIN {X 0,Y 190.947,Z 719.965,A -85,B 0,C 180,E1 7162.596,E2 7162.596} C_VEL
LIN {X 0,Y 181.064,Z 728.973,A -85,B 0,C 180,E1 7158.671,E2 7158.671} C_VEL
LIN {X 0,Y 170.368,Z 738.292,A -85,B 0,C 180,E1 7153.36,E2 7153.36} C_VEL
LIN {X 0,Y 159.979,Z 746.947,A -85,B 0,C 180,E1 7146.419,E2 7146.419} C_VEL
LIN {X 0,Y 153.31,Z 752.571,A -85,B 0,C 180,E1 7140.141,E2 7140.141} C_VEL
LIN {X 0,Y 148.66,Z 756.754,A -85,B 0,C 180,E1 7133.797,E2 7133.797} C_VEL
LIN {X 0,Y 145.66,Z 759.874,A -85,B 0,C 180,E1 7127.166,E2 7127.166} C_VEL
LIN {X 0,Y 144.327,Z 761.764,A -85,B 0,C 180,E1 7121.248,E2 7121.248} C_VEL
LIN {X 0,Y 143.052,Z 762.456,A -85,B 0,C 180,E1 7118.205,E2 7118.205} C_VEL
LIN {X 0,Y 139.599,Z 762.923,A -85,B 0,C 180,E1 7113.889,E2 7113.889} C_VEL
LIN {X 0,Y 136.19,Z 763.014,A -85,B 0,C 180,E1 7108.419,E2 7108.419} C_VEL
LIN {X 0,Y 135.974,Z 762.903,A -85,B 0,C 180,E1 7106.994,E2 7106.994} C_VEL
LIN {X 0,Y 136.118,Z 762.143,A -85,B 0,C 180,E1 7100.701,E2 7100.701} C_VEL
LIN {X 0,Y 137.515,Z 760.146,A -85,B 0,C 180,E1 7093.094,E2 7093.094} C_VEL
LIN {X 0,Y 140.526,Z 757.206,A -85,B 0,C 180,E1 7086.076,E2 7086.076} C_VEL
LIN {X 0,Y 145.368,Z 753.139,A -85,B 0,C 180,E1 7079.294,E2 7079.294} C_VEL
LIN {X 0,Y 151.727,Z 748.107,A -85,B 0,C 180,E1 7073.158,E2 7073.158} C_VEL
LIN {X 0,Y 159.718,Z 741.85,A -85,B 0,C 180,E1 7067.466,E2 7067.466} C_VEL
LIN {X 0,Y 169.077,Z 734.362,A -85,B 0,C 180,E1 7062.343,E2 7062.343} C_VEL
LIN {X 0,Y 181.587,Z 723.916,A -85,B 0,C 180,E1 7057.03,E2 7057.03} C_VEL
LIN {X 0,Y 194.844,Z 711.703,A -85,B 0,C 180,E1 7052.605,E2 7052.605} C_VEL
LIN {X 0,Y 205.794,Z 700.817,A -85,B 0,C 180,E1 7049.59,E2 7049.59} C_VEL
LIN {X 0,Y 215.83,Z 690.021,A -85,B 0,C 180,E1 7047.206,E2 7047.206} C_VEL
LIN {X 0,Y 226.21,Z 677.853,A -85,B 0,C 180,E1 7045.04,E2 7045.04} C_VEL
LIN {X 0,Y 236.309,Z 664.861,A -85,B 0,C 180,E1 7043.173,E2 7043.173} C_VEL
LIN {X 0,Y 246.15,Z 650.867,A -85,B 0,C 180,E1 7041.55,E2 7041.55} C_VEL
LIN {X 0,Y 255.961,Z 635.28,A -85,B 0,C 180,E1 7040.088,E2 7040.088} C_VEL
LIN {X 0,Y 267.352,Z 614.373,A -85,B 0,C 180,E1 7038.566,E2 7038.566} C_VEL
LIN {X 0,Y 275.314,Z 597.102,A -85,B 0,C 180,E1 7037.594,E2 7037.594} C_VEL
LIN {X 0,Y 282.02,Z 580.158,A -85,B 0,C 180,E1 7036.835,E2 7036.835} C_VEL
LIN {X 0,Y 287.426,Z 564.03,A -85,B 0,C 180,E1 7036.258,E2 7036.258} C_VEL
LIN {X 0,Y 292.205,Z 546.729,A -85,B 0,C 180,E1 7035.772,E2 7035.772} C_VEL
LIN {X 0,Y 296.029,Z 528.992,A -85,B 0,C 180,E1 7035.377,E2 7035.377} C_VEL
LIN {X 0,Y 299.097,Z 508.736,A -85,B 0,C 180,E1 7035.006,E2 7035.006} C_VEL
LIN {X 0,Y 308.305,Z 422.074,A -85,B 0,C 180,E1 7033.647,E2 7033.647} C_VEL
LIN {X 0,Y 305.46,Z 415.377,A -85,B 0,C 180,E1 7030.467,E2 7030.467} C_VEL
LIN {X 0,Y 303.618,Z 411.305,A -85,B 0,C 180,E1 7027.76,E2 7027.76} C_VEL
LIN {X 0,Y 302.381,Z 408.261,A -85,B 0,C 180,E1 7025.122,E2 7025.122} C_VEL
LIN {X 0,Y 301.399,Z 405.847,A -85,B 0,C 180,E1 7019.62,E2 7019.62} C_VEL
LIN {X 0,Y 302.595,Z 408.792,A -85,B 0,C 180,E1 7014.025,E2 7014.025} C_VEL
LIN {X 0,Y 304.363,Z 412.955,A -85,B 0,C 180,E1 7010.737,E2 7010.737} C_VEL
LIN {X 0,Y 306.759,Z 418.35,A -85,B 0,C 180,E1 7007.673,E2 7007.673} C_VEL
LIN {X 0,Y 309.782,Z 425.746,A -85,B 0,C 180,E1 7004.652,E2 7004.652} C_VEL
LIN {X 0,Y 313.405,Z 435.214,A -85,B 0,C 180,E1 7001.684,E2 7001.684} C_VEL
LIN {X 0,Y 321.472,Z 454.243,A -85,B 0,C 180,E1 6996.636,E2 6996.636} C_VEL
LIN {X 0,Y 332.37,Z 471.397,A -85,B 0,C 180,E1 6991.803,E2 6991.803} C_VEL
LIN {X 0,Y 344.978,Z 486.221,A -85,B 0,C 180,E1 6987.525,E2 6987.525} C_VEL
LIN {X 0,Y 369.618,Z 508.357,A -85,B 0,C 180,E1 6981.176,E2 6981.176} C_VEL
LIN {X 0,Y 387.14,Z 521.797,A -85,B 0,C 180,E1 6977.465,E2 6977.465} C_VEL
LIN {X 0,Y 397.625,Z 529.694,A -85,B 0,C 180,E1 6975.141,E2 6975.141} C_VEL
LIN {X 0,Y 407.634,Z 537.3,A -85,B 0,C 180,E1 6972.722,E2 6972.722} C_VEL
LIN {X 0,Y 417.439,Z 544.947,A -85,B 0,C 180,E1 6970.173,E2 6970.173} C_VEL
LIN {X 0,Y 425.964,Z 551.496,A -85,B 0,C 180,E1 6967.825,E2 6967.825} C_VEL
LIN {X 0,Y 434.949,Z 558.296,A -85,B 0,C 180,E1 6965.201,E2 6965.201} C_VEL
LIN {X 0,Y 443.268,Z 564.608,A -85,B 0,C 180,E1 6962.619,E2 6962.619} C_VEL
LIN {X 0,Y 449.163,Z 568.984,A -85,B 0,C 180,E1 6960.683,E2 6960.683} C_VEL
LIN {X 0,Y 455.768,Z 573.869,A -85,B 0,C 180,E1 6958.389,E2 6958.389} C_VEL
LIN {X 0,Y 461.574,Z 577.943,A -85,B 0,C 180,E1 6956.255,E2 6956.255} C_VEL
LIN {X 0,Y 467.725,Z 582.616,A -85,B 0,C 180,E1 6953.798,E2 6953.798} C_VEL
LIN {X 0,Y 474.292,Z 586.789,A -85,B 0,C 180,E1 6950.945,E2 6950.945} C_VEL
LIN {X 0,Y 479.363,Z 590.935,A -85,B 0,C 180,E1 6948.356,E2 6948.356} C_VEL
LIN {X 0,Y 484.128,Z 594.088,A -85,B 0,C 180,E1 6945.695,E2 6945.695} C_VEL
LIN {X 0,Y 488.359,Z 596.277,A -85,B 0,C 180,E1 6942.944,E2 6942.944} C_VEL
LIN {X 0,Y 490.678,Z 598.23,A -85,B 0,C 180,E1 6941.042,E2 6941.042} C_VEL
LIN {X 0,Y 493.268,Z 600.56,A -85,B 0,C 180,E1 6938.391,E2 6938.391} C_VEL
LIN {X 0,Y 495.206,Z 602.009,A -85,B 0,C 180,E1 6935.793,E2 6935.793} C_VEL
LIN {X 0,Y 496.485,Z 602.885,A -85,B 0,C 180,E1 6933.117,E2 6933.117} C_VEL
LIN {X 0,Y 496.98,Z 603.164,A -85,B 0,C 180,E1 6930.461,E2 6930.461} C_VEL
LIN {X 0,Y 496.754,Z 603.043,A -85,B 0,C 180,E1 6927.809,E2 6927.809} C_VEL
LIN {X 0,Y 495.714,Z 602.37,A -85,B 0,C 180,E1 6925.141,E2 6925.141} C_VEL
LIN {X 0,Y 494.067,Z 601.19,A -85,B 0,C 180,E1 6922.559,E2 6922.559} C_VEL
LIN {X 0,Y 491.626,Z 599.083,A -85,B 0,C 180,E1 6919.861,E2 6919.861} C_VEL
LIN {X 0,Y 488.629,Z 596.39,A -85,B 0,C 180,E1 6917.234,E2 6917.234} C_VEL
LIN {X 0,Y 484.486,Z 594.299,A -85,B 0,C 180,E1 6914.538,E2 6914.538} C_VEL
LIN {X 0,Y 480.147,Z 591.497,A -85,B 0,C 180,E1 6912.051,E2 6912.051} C_VEL
LIN {X 0,Y 474.869,Z 587.313,A -85,B 0,C 180,E1 6909.351,E2 6909.351} C_VEL
LIN {X 0,Y 469.272,Z 583.655,A -85,B 0,C 180,E1 6906.855,E2 6906.855} C_VEL
LIN {X 0,Y 462.784,Z 578.917,A -85,B 0,C 180,E1 6904.202,E2 6904.202} C_VEL
LIN {X 0,Y 457.344,Z 574.904,A -85,B 0,C 180,E1 6902.16,E2 6902.16} C_VEL
LIN {X 0,Y 450.573,Z 570.11,A -85,B 0,C 180,E1 6899.81,E2 6899.81} C_VEL
LIN {X 0,Y 444.232,Z 565.273,A -85,B 0,C 180,E1 6897.692,E2 6897.692} C_VEL
LIN {X 0,Y 435.894,Z 559.075,A -85,B 0,C 180,E1 6895.091,E2 6895.091} C_VEL
LIN {X 0,Y 427.994,Z 553.075,A -85,B 0,C 180,E1 6892.771,E2 6892.771} C_VEL
LIN {X 0,Y 418.684,Z 545.847,A -85,B 0,C 180,E1 6890.157,E2 6890.157} C_VEL
LIN {X 0,Y 409.309,Z 538.592,A -85,B 0,C 180,E1 6887.696,E2 6887.696} C_VEL
LIN {X 0,Y 398.699,Z 530.558,A -85,B 0,C 180,E1 6885.111,E2 6885.111} C_VEL
LIN {X 0,Y 388.021,Z 522.465,A -85,B 0,C 180,E1 6882.717,E2 6882.717} C_VEL
LIN {X 0,Y 370.134,Z 508.75,A -85,B 0,C 180,E1 6878.937,E2 6878.937} C_VEL
LIN {X 0,Y 345.461,Z 486.729,A -85,B 0,C 180,E1 6872.621,E2 6872.621} C_VEL
LIN {X 0,Y 332.757,Z 471.909,A -85,B 0,C 180,E1 6868.344,E2 6868.344} C_VEL
LIN {X 0,Y 321.797,Z 454.868,A -85,B 0,C 180,E1 6863.533,E2 6863.533} C_VEL
LIN {X 0,Y 313.638,Z 435.905,A -85,B 0,C 180,E1 6858.494,E2 6858.494} C_VEL
LIN {X 0,Y 310.39,Z 427.365,A -85,B 0,C 180,E1 6855.892,E2 6855.892} C_VEL
LIN {X 0,Y 307.607,Z 420.407,A -85,B 0,C 180,E1 6853.248,E2 6853.248} C_VEL
LIN {X 0,Y 304.947,Z 414.281,A -85,B 0,C 180,E1 6850.103,E2 6850.103} C_VEL
LIN {X 0,Y 303.548,Z 411.19,A -85,B 0,C 180,E1 6847.952,E2 6847.952} C_VEL
LIN {X 0,Y 302.331,Z 408.21,A -85,B 0,C 180,E1 6845.313,E2 6845.313} C_VEL
LIN {X 0,Y 301.399,Z 405.834,A -85,B 0,C 180,E1 6840,E2 6840} C_VEL
LIN {X 0,Y 302.571,Z 408.673,A -85,B 0,C 180,E1 6834.405,E2 6834.405} C_VEL
LIN {X 0,Y 304.376,Z 412.994,A -85,B 0,C 180,E1 6831.023,E2 6831.023} C_VEL
LIN {X 0,Y 306.609,Z 418.047,A -85,B 0,C 180,E1 6828.144,E2 6828.144} C_VEL
LIN {X 0,Y 308.315,Z 422.305,A -85,B 0,C 180,E1 6826.323,E2 6826.323} C_VEL
LIN {X 0,Y 298.082,Z 516.509,A -85,B 0,C 180,E1 6824.862,E2 6824.862} C_VEL
LIN {X 0,Y 293.951,Z 539.719,A -85,B 0,C 180,E1 6824.398,E2 6824.398} C_VEL
LIN {X 0,Y 288.333,Z 561.059,A -85,B 0,C 180,E1 6823.833,E2 6823.833} C_VEL
LIN {X 0,Y 282.917,Z 577.672,A -85,B 0,C 180,E1 6823.264,E2 6823.264} C_VEL
LIN {X 0,Y 276.648,Z 593.917,A -85,B 0,C 180,E1 6822.562,E2 6822.562} C_VEL
LIN {X 0,Y 269.554,Z 609.774,A -85,B 0,C 180,E1 6821.71,E2 6821.71} C_VEL
LIN {X 0,Y 261.654,Z 625.21,A -85,B 0,C 180,E1 6820.693,E2 6820.693} C_VEL
LIN {X 0,Y 252.989,Z 640.183,A -85,B 0,C 180,E1 6819.483,E2 6819.483} C_VEL
LIN {X 0,Y 242.768,Z 655.906,A -85,B 0,C 180,E1 6817.908,E2 6817.908} C_VEL
LIN {X 0,Y 228.964,Z 674.478,A -85,B 0,C 180,E1 6815.489,E2 6815.489} C_VEL
LIN {X 0,Y 218.197,Z 687.353,A -85,B 0,C 180,E1 6813.312,E2 6813.312} C_VEL
LIN {X 0,Y 207.313,Z 699.234,A -85,B 0,C 180,E1 6810.793,E2 6810.793} C_VEL
LIN {X 0,Y 196.882,Z 709.725,A -85,B 0,C 180,E1 6807.996,E2 6807.996} C_VEL
LIN {X 0,Y 186.291,Z 719.613,A -85,B 0,C 180,E1 6804.659,E2 6804.659} C_VEL
LIN {X 0,Y 175.773,Z 728.794,A -85,B 0,C 180,E1 6800.672,E2 6800.672} C_VEL
LIN {X 0,Y 164.517,Z 738.114,A -85,B 0,C 180,E1 6795.316,E2 6795.316} C_VEL
LIN {X 0,Y 153.476,Z 746.768,A -85,B 0,C 180,E1 6788.231,E2 6788.231} C_VEL
LIN {X 0,Y 146.303,Z 752.393,A -85,B 0,C 180,E1 6781.747,E2 6781.747} C_VEL
LIN {X 0,Y 141.095,Z 756.701,A -85,B 0,C 180,E1 6774.893,E2 6774.893} C_VEL
LIN {X 0,Y 137.779,Z 759.846,A -85,B 0,C 180,E1 6767.744,E2 6767.744} C_VEL
LIN {X 0,Y 136.238,Z 761.873,A -85,B 0,C 180,E1 6760.571,E2 6760.571} C_VEL
LIN {X 0,Y 135.963,Z 762.816,A -85,B 0,C 180,E1 6754.217,E2 6754.217} C_VEL
LIN {X 0,Y 135.996,Z 762.997,A -85,B 0,C 180,E1 6748.315,E2 6748.315} C_VEL
LIN {X 0,Y 135.974,Z 762.903,A -85,B 0,C 180,E1 6746.994,E2 6746.994} C_VEL
LIN {X 0,Y 135.103,Z 762.69,A -85,B 0,C 180,E1 6743.977,E2 6743.977} C_VEL
LIN {X 0,Y 131.925,Z 761.828,A -85,B 0,C 180,E1 6739.131,E2 6739.131} C_VEL
LIN {X 0,Y 129.632,Z 760.638,A -85,B 0,C 180,E1 6734.07,E2 6734.07} C_VEL
LIN {X 0,Y 129.83,Z 759.905,A -85,B 0,C 180,E1 6731.863,E2 6731.863} C_VEL
LIN {X 0,Y 133.376,Z 756.818,A -85,B 0,C 180,E1 6724.23,E2 6724.23} C_VEL
LIN {X 0,Y 138.681,Z 752.757,A -85,B 0,C 180,E1 6717.27,E2 6717.27} C_VEL
LIN {X 0,Y 145.818,Z 747.527,A -85,B 0,C 180,E1 6710.792,E2 6710.792} C_VEL
LIN {X 0,Y 154.888,Z 740.871,A -85,B 0,C 180,E1 6704.764,E2 6704.764} C_VEL
LIN {X 0,Y 167.463,Z 731.324,A -85,B 0,C 180,E1 6698.55,E2 6698.55} C_VEL
LIN {X 0,Y 180.456,Z 720.513,A -85,B 0,C 180,E1 6693.648,E2 6693.648} C_VEL
LIN {X 0,Y 191.933,Z 710.248,A -85,B 0,C 180,E1 6690.155,E2 6690.155} C_VEL
LIN {X 0,Y 202.679,Z 699.847,A -85,B 0,C 180,E1 6687.391,E2 6687.391} C_VEL
LIN {X 0,Y 213.044,Z 688.954,A -85,B 0,C 180,E1 6685.084,E2 6685.084} C_VEL
LIN {X 0,Y 224.016,Z 676.333,A -85,B 0,C 180,E1 6682.943,E2 6682.943} C_VEL
LIN {X 0,Y 234.694,Z 662.776,A -85,B 0,C 180,E1 6681.108,E2 6681.108} C_VEL
LIN {X 0,Y 247.226,Z 644.961,A -85,B 0,C 180,E1 6679.214,E2 6679.214} C_VEL
LIN {X 0,Y 258.21,Z 626.644,A -85,B 0,C 180,E1 6677.735,E2 6677.735} C_VEL
LIN {X 0,Y 266.687,Z 610.518,A -85,B 0,C 180,E1 6676.701,E2 6676.701} C_VEL
LIN {X 0,Y 273.763,Z 595.108,A -85,B 0,C 180,E1 6675.898,E2 6675.898} C_VEL
LIN {X 0,Y 280.253,Z 578.739,A -85,B 0,C 180,E1 6675.212,E2 6675.212} C_VEL
LIN {X 0,Y 285.673,Z 562.592,A -85,B 0,C 180,E1 6674.673,E2 6674.673} C_VEL
LIN {X 0,Y 290.543,Z 544.908,A -85,B 0,C 180,E1 6674.21,E2 6674.21} C_VEL
LIN {X 0,Y 295.056,Z 523.37,A -85,B 0,C 180,E1 6673.762,E2 6673.762} C_VEL
LIN {X 0,Y 298.96,Z 492.103,A -85,B 0,C 180,E1 6673.26,E2 6673.26} C_VEL
LIN {X 0,Y 305.906,Z 427.43,A -85,B 0,C 180,E1 6672.267,E2 6672.267} C_VEL
LIN {X 0,Y 303.496,Z 421.575,A -85,B 0,C 180,E1 6669.195,E2 6669.195} C_VEL
LIN {X 0,Y 302.307,Z 418.793,A -85,B 0,C 180,E1 6667.22,E2 6667.22} C_VEL
LIN {X 0,Y 301.251,Z 416.051,A -85,B 0,C 180,E1 6664.76,E2 6664.76} C_VEL
LIN {X 0,Y 300.422,Z 413.802,A -85,B 0,C 180,E1 6659.619,E2 6659.619} C_VEL
LIN {X 0,Y 301.492,Z 416.605,A -85,B 0,C 180,E1 6654.29,E2 6654.29} C_VEL
LIN {X 0,Y 303.177,Z 420.803,A -85,B 0,C 180,E1 6650.987,E2 6650.987} C_VEL
LIN {X 0,Y 305.37,Z 426.03,A -85,B 0,C 180,E1 6648.047,E2 6648.047} C_VEL
LIN {X 0,Y 308.13,Z 433.15,A -85,B 0,C 180,E1 6645.146,E2 6645.146} C_VEL
LIN {X 0,Y 311.373,Z 442.127,A -85,B 0,C 180,E1 6642.334,E2 6642.334} C_VEL
LIN {X 0,Y 319.216,Z 461.285,A -85,B 0,C 180,E1 6637.193,E2 6637.193} C_VEL
LIN {X 0,Y 329.835,Z 478.38,A -85,B 0,C 180,E1 6632.317,E2 6632.317} C_VEL
LIN {X 0,Y 342.376,Z 493.364,A -85,B 0,C 180,E1 6627.941,E2 6627.941} C_VEL
LIN {X 0,Y 366.405,Z 515.357,A -85,B 0,C 180,E1 6621.523,E2 6621.523} C_VEL
LIN {X 0,Y 385.756,Z 530.394,A -85,B 0,C 180,E1 6617.276,E2 6617.276} C_VEL
LIN {X 0,Y 395.614,Z 537.862,A -85,B 0,C 180,E1 6615.055,E2 6615.055} C_VEL
LIN {X 0,Y 406.043,Z 545.714,A -85,B 0,C 180,E1 6612.531,E2 6612.531} C_VEL
LIN {X 0,Y 415.502,Z 553.018,A -85,B 0,C 180,E1 6610.07,E2 6610.07} C_VEL
LIN {X 0,Y 425.264,Z 560.518,A -85,B 0,C 180,E1 6607.371,E2 6607.371} C_VEL
LIN {X 0,Y 433.145,Z 566.52,A -85,B 0,C 180,E1 6605.045,E2 6605.045} C_VEL
LIN {X 0,Y 440.837,Z 572.253,A -85,B 0,C 180,E1 6602.666,E2 6602.666} C_VEL
LIN {X 0,Y 446.727,Z 576.636,A -85,B 0,C 180,E1 6600.74,E2 6600.74} C_VEL
LIN {X 0,Y 454.452,Z 582.204,A -85,B 0,C 180,E1 6598.08,E2 6598.08} C_VEL
LIN {X 0,Y 459.733,Z 586.025,A -85,B 0,C 180,E1 6596.12,E2 6596.12} C_VEL
LIN {X 0,Y 466.399,Z 590.947,A -85,B 0,C 180,E1 6593.426,E2 6593.426} C_VEL
LIN {X 0,Y 472.311,Z 594.759,A -85,B 0,C 180,E1 6590.831,E2 6590.831} C_VEL
LIN {X 0,Y 477.515,Z 598.914,A -85,B 0,C 180,E1 6588.177,E2 6588.177} C_VEL
LIN {X 0,Y 482.216,Z 601.959,A -85,B 0,C 180,E1 6585.513,E2 6585.513} C_VEL
LIN {X 0,Y 486.261,Z 604.005,A -85,B 0,C 180,E1 6582.92,E2 6582.92} C_VEL
LIN {X 0,Y 489.265,Z 606.617,A -85,B 0,C 180,E1 6580.359,E2 6580.359} C_VEL
LIN {X 0,Y 491.651,Z 608.724,A -85,B 0,C 180,E1 6577.713,E2 6577.713} C_VEL
LIN {X 0,Y 493.467,Z 610.019,A -85,B 0,C 180,E1 6574.998,E2 6574.998} C_VEL
LIN {X 0,Y 494.466,Z 610.68,A -85,B 0,C 180,E1 6572.434,E2 6572.434} C_VEL
LIN {X 0,Y 494.805,Z 610.858,A -85,B 0,C 180,E1 6569.884,E2 6569.884} C_VEL
LIN {X 0,Y 494.455,Z 610.647,A -85,B 0,C 180,E1 6567.405,E2 6567.405} C_VEL
LIN {X 0,Y 493.354,Z 609.928,A -85,B 0,C 180,E1 6564.768,E2 6564.768} C_VEL
LIN {X 0,Y 491.662,Z 608.73,A -85,B 0,C 180,E1 6562.287,E2 6562.287} C_VEL
LIN {X 0,Y 489.111,Z 606.498,A -85,B 0,C 180,E1 6559.518,E2 6559.518} C_VEL
LIN {X 0,Y 486.232,Z 603.991,A -85,B 0,C 180,E1 6557.049,E2 6557.049} C_VEL
LIN {X 0,Y 482.219,Z 601.959,A -85,B 0,C 180,E1 6554.488,E2 6554.488} C_VEL
LIN {X 0,Y 477.5,Z 598.91,A -85,B 0,C 180,E1 6551.822,E2 6551.822} C_VEL
LIN {X 0,Y 472.525,Z 594.948,A -85,B 0,C 180,E1 6549.277,E2 6549.277} C_VEL
LIN {X 0,Y 468.159,Z 592.072,A -85,B 0,C 180,E1 6547.319,E2 6547.319} C_VEL
LIN {X 0,Y 461.769,Z 587.642,A -85,B 0,C 180,E1 6544.685,E2 6544.685} C_VEL
LIN {X 0,Y 455.561,Z 582.93,A -85,B 0,C 180,E1 6542.329,E2 6542.329} C_VEL
LIN {X 0,Y 447.636,Z 577.349,A -85,B 0,C 180,E1 6539.566,E2 6539.566} C_VEL
LIN {X 0,Y 441.687,Z 572.837,A -85,B 0,C 180,E1 6537.608,E2 6537.608} C_VEL
LIN {X 0,Y 434.686,Z 567.758,A -85,B 0,C 180,E1 6535.436,E2 6535.436} C_VEL
LIN {X 0,Y 426.932,Z 561.757,A -85,B 0,C 180,E1 6533.112,E2 6533.112} C_VEL
LIN {X 0,Y 417.466,Z 554.415,A -85,B 0,C 180,E1 6530.465,E2 6530.465} C_VEL
LIN {X 0,Y 408.222,Z 547.485,A -85,B 0,C 180,E1 6528.021,E2 6528.021} C_VEL
LIN {X 0,Y 397.947,Z 539.693,A -85,B 0,C 180,E1 6525.499,E2 6525.499} C_VEL
LIN {X 0,Y 388.467,Z 532.411,A -85,B 0,C 180,E1 6523.311,E2 6523.311} C_VEL
LIN {X 0,Y 376.003,Z 523.035,A -85,B 0,C 180,E1 6520.656,E2 6520.656} C_VEL
LIN {X 0,Y 355.158,Z 505.723,A -85,B 0,C 180,E1 6515.696,E2 6515.696} C_VEL
LIN {X 0,Y 334.737,Z 484.838,A -85,B 0,C 180,E1 6509.529,E2 6509.529} C_VEL
LIN {X 0,Y 322.185,Z 466.683,A -85,B 0,C 180,E1 6504.33,E2 6504.33} C_VEL
LIN {X 0,Y 313.365,Z 447.899,A -85,B 0,C 180,E1 6499.187,E2 6499.187} C_VEL
LIN {X 0,Y 309.688,Z 437.384,A -85,B 0,C 180,E1 6496.266,E2 6496.266} C_VEL
LIN {X 0,Y 306.573,Z 429.06,A -85,B 0,C 180,E1 6493.293,E2 6493.293} C_VEL
LIN {X 0,Y 304.017,Z 422.697,A -85,B 0,C 180,E1 6490.23,E2 6490.23} C_VEL
LIN {X 0,Y 302.346,Z 418.887,A -85,B 0,C 180,E1 6487.602,E2 6487.602} C_VEL
LIN {X 0,Y 301.279,Z 416.092,A -85,B 0,C 180,E1 6485.141,E2 6485.141} C_VEL
LIN {X 0,Y 300.423,Z 413.784,A -85,B 0,C 180,E1 6480,E2 6480} C_VEL
LIN {X 0,Y 301.502,Z 416.611,A -85,B 0,C 180,E1 6474.576,E2 6474.576} C_VEL
LIN {X 0,Y 303.131,Z 420.689,A -85,B 0,C 180,E1 6471.368,E2 6471.368} C_VEL
LIN {X 0,Y 305.269,Z 425.783,A -85,B 0,C 180,E1 6468.474,E2 6468.474} C_VEL
LIN {X 0,Y 305.918,Z 427.656,A -85,B 0,C 180,E1 6467.699,E2 6467.699} C_VEL
LIN {X 0,Y 296.073,Z 516.455,A -85,B 0,C 180,E1 6466.358,E2 6466.358} C_VEL
LIN {X 0,Y 291.825,Z 539.826,A -85,B 0,C 180,E1 6465.908,E2 6465.908} C_VEL
LIN {X 0,Y 286.203,Z 560.884,A -85,B 0,C 180,E1 6465.376,E2 6465.376} C_VEL
LIN {X 0,Y 280.708,Z 577.497,A -85,B 0,C 180,E1 6464.835,E2 6464.835} C_VEL
LIN {X 0,Y 274.05,Z 594.434,A -85,B 0,C 180,E1 6464.133,E2 6464.133} C_VEL
LIN {X 0,Y 267.136,Z 609.598,A -85,B 0,C 180,E1 6463.351,E2 6463.351} C_VEL
LIN {X 0,Y 259.099,Z 625.033,A -85,B 0,C 180,E1 6462.377,E2 6462.377} C_VEL
LIN {X 0,Y 250.27,Z 640.007,A -85,B 0,C 180,E1 6461.216,E2 6461.216} C_VEL
LIN {X 0,Y 239.84,Z 655.729,A -85,B 0,C 180,E1 6459.7,E2 6459.7} C_VEL
